// TIA Portal project "Inteligenta_szklarnia" (V15.1)

(* hardware
DEVICE "S7-1200 station_2"  S7-1200 Station
   slot 0: "Rack_0"  S7-1200 Rack  Rack  V1.0
   slot 1: "PLC_1"  CPU 1214C AC/DC/Rly  6ES7 214-1BE30-0XB0  V2.2
DEVICE "HMI_1"  KTP700 Basic PN
   slot 0: "HMI_1"  KTP700 Basic PN  6AV2 123-2GB03-0AX0  15.0.0.0
   slot 1: "HMI_RT_3"  KTP700 Basic PN  6AV2 123-2GB03-0AX0  15.0.0.0
   slot 5: "HMI_1.IE_CP_1"  PROFINET Interface  15.0.0.0
      slot 1: "PROFINET Interface_1"  PROFINET Interface
         slot 1: "Port_1"  Port
DEVICE "S7-1200 station_1"  S7-1200 Station
   slot 0: "Rack_0"  S7-1200 Rack  Rack  V1.0
   slot 1: "PLC_do_symulacji"  CPU 1214C AC/DC/Rly  6ES7 214-1BG40-0XB0  V4.2
DEVICE "HMI_do_symulacji"  KTP700 Basic PN
   slot 0: "HMI_do_symulacji"  KTP700 Basic PN  6AV2 123-2GB03-0AX0  15.1.0.0
   slot 1: "HMI_RT_2"  KTP700 Basic PN  6AV2 123-2GB03-0AX0  15.1.0.0
   slot 5: "HMI_do_symulacji.IE_CP_1"  PROFINET Interface  15.0.1.0
      slot 1: "PROFINET Interface_1"  PROFINET Interface
         slot 1: "Port_1"  Port
DEVICE "S71500/ET200MP station_1"  S7-1500 station
   slot 0: "Rail_0"  Rack  6ES7 590-1***0-0AA0
   slot 1: "PLC_Web_server"  CPU 1518-4 PN/DP  6ES7 518-4AP00-0AB0  V2.6
      slot 3: "CPU display_1"  6ES7591-1BA00-0AA0
*)

// ===== PLC "PLC_1"  CPU 1214C AC/DC/Rly =====

VAR_GLOBAL   // PLC tag table "Default tag table"
   "Tag_1" AT %M0.0 : Bool;
   "System_Byte" AT %MB1 : Byte;
   "FirstScan" AT %M1.0 : Bool;
   "DiagStatusUpdate" AT %M1.1 : Bool;
   "AlwaysTRUE" AT %M1.2 : Bool;
   "AlwaysFALSE" AT %M1.3 : Bool;
   "Tag_2" AT %M0.1 : Bool;
   "Clock_Byte" AT %MB30 : Byte;
   "Clock_10Hz" AT %M30.0 : Bool;
   "Clock_5Hz" AT %M30.1 : Bool;
   "Clock_2.5Hz" AT %M30.2 : Bool;
   "Clock_2Hz" AT %M30.3 : Bool;
   "Clock_1.25Hz" AT %M30.4 : Bool;
   "Clock_1Hz" AT %M30.5 : Bool;
   "Clock_0.625Hz" AT %M30.6 : Bool;
   "Clock_0.5Hz" AT %M30.7 : Bool;
   "marker_clock" AT %M0.2 : Bool;
   "marker_counter" AT %M0.3 : Bool;
   "wartosc_rolet_sym" AT %MW2 : Int;
   "swiatlo_bez_rolet" AT %MW4 : Int;
   "Alarm_active" AT %M8.0 : Bool;
   "Clock_Byte(1)" AT %MB0 : Byte;
   "Clock_10Hz(1)" AT %M0.0 : Bool;
   "Clock_5Hz(1)" AT %M0.1 : Bool;
   "Clock_2.5Hz(1)" AT %M0.2 : Bool;
   "Clock_2Hz(1)" AT %M0.3 : Bool;
   "Clock_1.25Hz(1)" AT %M0.4 : Bool;
   "Clock_1Hz(1)" AT %M0.5 : Bool;
   "Clock_0.625Hz(1)" AT %M0.6 : Bool;
   "Clock_0.5Hz(1)" AT %M0.7 : Bool;
END_VAR

VAR_GLOBAL   // PLC tag table "wyjscia"
   "Grzałka" AT %Q0.0 : Bool;
   "Wentylator" AT %Q0.1 : Bool;
   "Pompa_zraszacze" AT %Q0.2 : Bool;   // Pompa zraszaczy, które odpowiadają za wilgotność powietrza w szklarni
   "Rolety_zamykanie" AT %Q0.4 : Bool;
   "Alarm_ostrzegwaczy" AT %Q0.5 : Bool;
   "Siłownik_okien_otwieranie" AT %Q0.6 : Bool;
   "Siłownik_okien_zamykanie" AT %Q0.7 : Bool;
   "Rolety_otwieranie" AT %Q0.3 : Bool;
   "Pompa_podlewanie" AT %Q1.0 : Bool;   // Pompa podlewania kropelkowego, która odpowiada za wilgotność gleby
END_VAR

DATA_BLOCK "Wejscia_PLC"   // DB1
{ S7_Optimized_Access := 'TRUE' }
VERSION : 0.1
   VAR
      Czujnik_wilgotności_powietrza : Int;   // Czujnik wilgotności powietrza w szklarni
      Czujnik_wilgotności_gleby : Int;   // Czujnik wilgotności gleby w szklarni
      Temperatura_wewnetrzna : Real;   // Temperatura wewnątrz szklarni
      Czujnik_natezenia_swiatła : Int;   // Czujnik natężenia światła wewnątrz szklarni
      Czujnik_wiatru : Int;   // Czujnik prędkości wiatru poza szklarnią
      Wewnetrzny_czujnik_CO2 : Int;   // Czujnik stężenia dwutlenku węgla w szklarni
      Stopien_zasloniecia_rolet : Int;   // Stopień zasłonięcia rolet w szklarni (przyjęty przedział 0-100%)
      Temperatura_zewnetrzna : Real;   // Temperatura mierzona na zewnątrz, poza szklarnią. Typ Int, ponieważ nie jest wymagana taka dokładność jak w pomiarze temperatury wewnętrznej.
      Zewnetrzny_czujnik_CO2 : Int;   // Czujnik stężenia dwutlenku węgla poza szklarnią
      czujnik_wilgotnosci_zewnetrzny : Int := 50;   // Potrzebny w ramach symulacji realnych warunkow
   END_VAR
BEGIN
END_DATA_BLOCK

DATA_BLOCK "HMI"   // DB2
{ S7_Optimized_Access := 'TRUE' }
VERSION : 0.1
   VAR
      nazwa_receptury : String;
      System_okien_auto : Bool;   // Wł/wył system okien w trybie automatycznym
      Przycisk_zraszacze_manual : Bool;   // Przycisk pompy zraszaczy w trybie manualnym
      Przycisk_podlewanie_manual : Bool;   // Przycisk pompy podlewania w trybie manualnym
      Przycisk_grzanie_manual : Bool;   // Przycisk grzałki w trybie manualnym
      Przycisk_wentylacja_manual : Bool;   // Przycisk wentylacji w trybie manualnym
      Otwarcie_okien_manual : Bool;   // Ustawiony w trybie manualnym otwarcie okien
      Stopien_zasloniecia_rolet_manual : Int;   // Ustawiony w trybie manualnym stopień zasłonięcia rolet
      Temperatura_auto : Real := 22.0;   // Nastawiona temeratura w trybie automatycznym
      Naslonecznienie_auto : Int := 1000;   // Nastawiona wartość nasłonecznienia w trybie automatycznym
      Wilgotnosc_powietrza_auto : Int := 50;   // Nastawiona wartość wilgotności powietrza w trybie automatycznym
      Poziom_CO2_auto : Int := 800;   // Nastawiona wartość stężenia CO2 w trybie automatycznym
      Wilgotnosc_gleby_auto : Int := 60;   // Nastawiona wartość wilgotności gleby w trybie automatycznym
      Przycisk_zatwierdz_auto : Bool;   // Przycisk zatwierdzający wcześniej wybrane ustawienia trybu automatycznego
      Przycisk_zatwierdz_zapis_receptury : Bool;   // Przycisk zatwierdzający wcześniej wybrane ustawienia trybu zapisania receptury
      Przycisk_zatwierdz_wybor_receptury : Bool;   // Przycisk zatwierdzający wcześniej wybrane ustawienia trybu receptury
      Numer_ekranu_HMI : Int;   // Numer aktualnie otwartego ekranu w HMI
      Aktywacja_trybu_manualnego : Bool;
      Aktywacja_trybu_automatycznego : Bool;
      Aktywacja_trybu_Receptur : Bool;
      Aktywacja_trybu_zapis_Receptur : Bool;
      Reset_Trybow : Bool;
   END_VAR
BEGIN
END_DATA_BLOCK

DATA_BLOCK "Tryb_auto_parametry"   // DB7
{ S7_Optimized_Access := 'TRUE' }
VERSION : 0.1
   VAR
      Temperatura : Real;
      Naslonecznienie : Int;
      Wilgotnosc_powietrza : Int;
      Wilgotnosc_gleby : Int;
      System_okien : Bool;
      Stezenie_co2 : Int;
   END_VAR
BEGIN
END_DATA_BLOCK

DATA_BLOCK "Alarmy"   // DB9
{ S7_Optimized_Access := 'TRUE' }
VERSION : 0.1
   VAR
      Warning_niska_temp_1 : Bool;
      Warning_wysoka_temp_1 : Bool;
      Warning_nieprawidlowe_CO2_1 : Bool;
      Blad_zbyt_wysokie_CO2_1 : Bool;
   END_VAR
BEGIN
END_DATA_BLOCK

// folder: Archiwizacja_parametrow

DATA_BLOCK "Archiwizowane_parametry"   // DB4
{ S7_Optimized_Access := 'TRUE' }
VERSION : 0.1
   VAR
      Temperatura : Array[0..111] of Real;
      Wilgotnosc : Array[0..111] of Int;
      Naslonecznienie : Array[0..111] of Int;
      iterator : Int := 0;   // Iterator służący do zapisu danych w odpowiednich komórkach tablicy.
   END_VAR
BEGIN
   Naslonecznienie[0] := 0;
   Naslonecznienie[1] := 0;
END_DATA_BLOCK

// folder: System blocks/Program resources

DATA_BLOCK "IEC_Counter_0_DB_1"   // DB3
{ S7_Optimized_Access := 'TRUE' }
AUTHOR : Simatic
FAMILY : IEC
NAME : CNTR
VERSION : 1.0
// stored: InstanceOfName IEC_COUNTER
"IEC_COUNTER"
BEGIN
END_DATA_BLOCK

DATA_BLOCK "IEC_Timer_0_DB"   // DB5
{ S7_Optimized_Access := 'TRUE' }
AUTHOR : Simatic
FAMILY : IEC
NAME : IEC_TMR
VERSION : 1.0
// stored: InstanceOfName IEC_TIMER
"IEC_TIMER"
BEGIN
END_DATA_BLOCK

DATA_BLOCK "IEC_Timer_0_DB_1"   // DB6
{ S7_Optimized_Access := 'TRUE' }
AUTHOR : Simatic
FAMILY : IEC
NAME : IEC_TMR
VERSION : 1.0
// stored: InstanceOfName IEC_TIMER
"IEC_TIMER"
BEGIN
END_DATA_BLOCK

DATA_BLOCK "IEC_Timer_0_DB_2"   // DB8
{ S7_Optimized_Access := 'TRUE' }
AUTHOR : Simatic
FAMILY : IEC
NAME : IEC_TMR
VERSION : 1.0
// stored: InstanceOfName IEC_TIMER
"IEC_TIMER"
BEGIN
END_DATA_BLOCK

DATA_BLOCK "IEC_Timer_0_DB_5"   // DB10
{ S7_Optimized_Access := 'TRUE' }
AUTHOR : Simatic
FAMILY : IEC
NAME : IEC_TMR
VERSION : 1.0
// stored: InstanceOfName IEC_TIMER
"IEC_TIMER"
BEGIN
END_DATA_BLOCK

DATA_BLOCK "IEC_Timer_0_DB_3"   // DB11
{ S7_Optimized_Access := 'TRUE' }
AUTHOR : Simatic
FAMILY : IEC
NAME : IEC_TMR
VERSION : 1.0
// stored: InstanceOfName IEC_TIMER
"IEC_TIMER"
BEGIN
END_DATA_BLOCK

DATA_BLOCK "IEC_Counter_0_DB"   // DB12
{ S7_Optimized_Access := 'TRUE' }
AUTHOR : Simatic
FAMILY : IEC
NAME : CNTR
VERSION : 1.0
// stored: InstanceOfName IEC_COUNTER
"IEC_COUNTER"
BEGIN
END_DATA_BLOCK

DATA_BLOCK "IEC_Counter_0_DB_2"   // DB13
{ S7_Optimized_Access := 'TRUE' }
AUTHOR : Simatic
FAMILY : IEC
NAME : CNTR
VERSION : 1.0
// stored: InstanceOfName IEC_COUNTER
"IEC_COUNTER"
BEGIN
END_DATA_BLOCK

// folder: (top level)

FUNCTION "Rolety" : Void   // FC1, LAD
{ S7_Optimized_Access := 'TRUE' }
VERSION : 0.1
   VAR_INPUT
      Czy_automatyczny : Bool;
      Czy_manualny : Bool;
   END_VAR
BEGIN

REGION Network 1: Warunki otwierania rolet w trybie automatycznym i manualnym
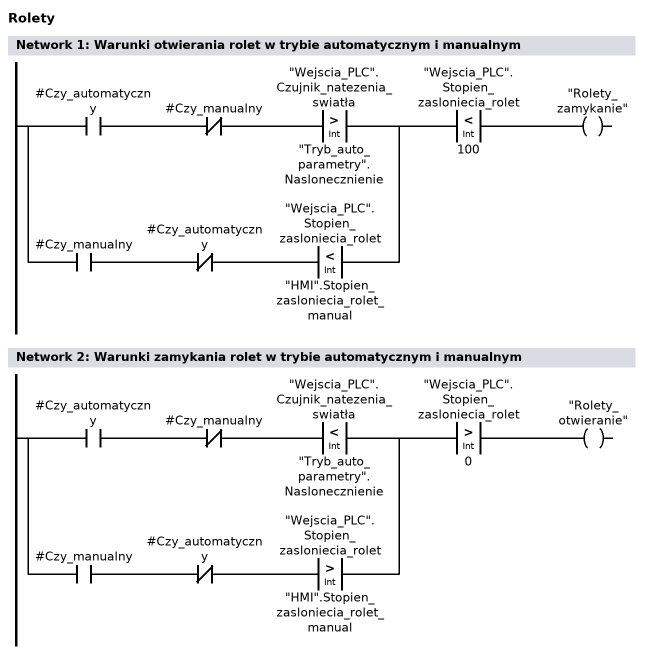
   RUNG wire#powerrail
      Contact( #Czy_automatyczny )
      I_Contact( #Czy_manualny )
      { S7_Templates := "SrcType := Int" } GT_Contact(in1 := "Wejscia_PLC".Czujnik_natezenia_swiatła, in2 := "Tryb_auto_parametry".Naslonecznienie)
      wire#w1
      { S7_Templates := "SrcType := Int" } LT_Contact(in1 := "Wejscia_PLC".Stopien_zasloniecia_rolet, in2 := 100)
      Coil( "Rolety_zamykanie" )
   END_RUNG
   RUNG wire#powerrail
      Contact( #Czy_manualny )
      I_Contact( #Czy_automatyczny )
      { S7_Templates := "SrcType := Int" } LT_Contact(in1 := "Wejscia_PLC".Stopien_zasloniecia_rolet, in2 := "HMI".Stopien_zasloniecia_rolet_manual)
   END_RUNG wire#w1
   // the same network as SCL:
   "Rolety_zamykanie" := ((#Czy_automatyczny AND NOT #Czy_manualny AND ("Wejscia_PLC".Czujnik_natezenia_swiatła > "Tryb_auto_parametry".Naslonecznienie)) OR (#Czy_manualny AND NOT #Czy_automatyczny AND ("Wejscia_PLC".Stopien_zasloniecia_rolet < "HMI".Stopien_zasloniecia_rolet_manual))) AND ("Wejscia_PLC".Stopien_zasloniecia_rolet < 100);
END_REGION

REGION Network 2: Warunki zamykania rolet w trybie automatycznym i manualnym
   RUNG wire#powerrail
      Contact( #Czy_automatyczny )
      I_Contact( #Czy_manualny )
      { S7_Templates := "SrcType := Int" } LT_Contact(in1 := "Wejscia_PLC".Czujnik_natezenia_swiatła, in2 := "Tryb_auto_parametry".Naslonecznienie)
      wire#w1
      { S7_Templates := "SrcType := Int" } GT_Contact(in1 := "Wejscia_PLC".Stopien_zasloniecia_rolet, in2 := 0)
      Coil( "Rolety_otwieranie" )
   END_RUNG
   RUNG wire#powerrail
      Contact( #Czy_manualny )
      I_Contact( #Czy_automatyczny )
      { S7_Templates := "SrcType := Int" } GT_Contact(in1 := "Wejscia_PLC".Stopien_zasloniecia_rolet, in2 := "HMI".Stopien_zasloniecia_rolet_manual)
   END_RUNG wire#w1
   // the same network as SCL:
   "Rolety_otwieranie" := ((#Czy_automatyczny AND NOT #Czy_manualny AND ("Wejscia_PLC".Czujnik_natezenia_swiatła < "Tryb_auto_parametry".Naslonecznienie)) OR (#Czy_manualny AND NOT #Czy_automatyczny AND ("Wejscia_PLC".Stopien_zasloniecia_rolet > "HMI".Stopien_zasloniecia_rolet_manual))) AND ("Wejscia_PLC".Stopien_zasloniecia_rolet > 0);
END_REGION
END_FUNCTION

FUNCTION "Sterowanie_grzalka_wentylator" : Void   // FC3, LAD
{ S7_Optimized_Access := 'TRUE' }
VERSION : 0.1
   VAR_INPUT
      czy_manualny : Bool;
      czy_automatyczny : Bool;
   END_VAR
   VAR_TEMP
      Histereza_minus : Real;   // Wartość zadanej temperatury zmieniona o dolną wartość hiterezy
      Histereza_plus : Real;   // Wartość zadanej temperatury zmieniona o górną wartość hiterezy
   END_VAR
   VAR CONSTANT
      Wartosc_histerezy : Real := 1.0;
   END_VAR
   VAR_TEMP   // added for the SCL form of the ladder/FBD networks
      _w1 : Bool;
   END_VAR
BEGIN

REGION Network 1: Sterowanie wentylatorem w trybie automatycznym i manualnym
   // Gdy uruchomiony jest tryb automatyczny, wartość temperatury w szklarni powinna się mieścić w zakresie temperatury nastawionej +- wartość histerezy. Gdy jest ona za wysoka uruchamiany jest wentylator. W trybie manualnym włączany jest on od razu po naciśnięciu przycisku do niego przypisanego.
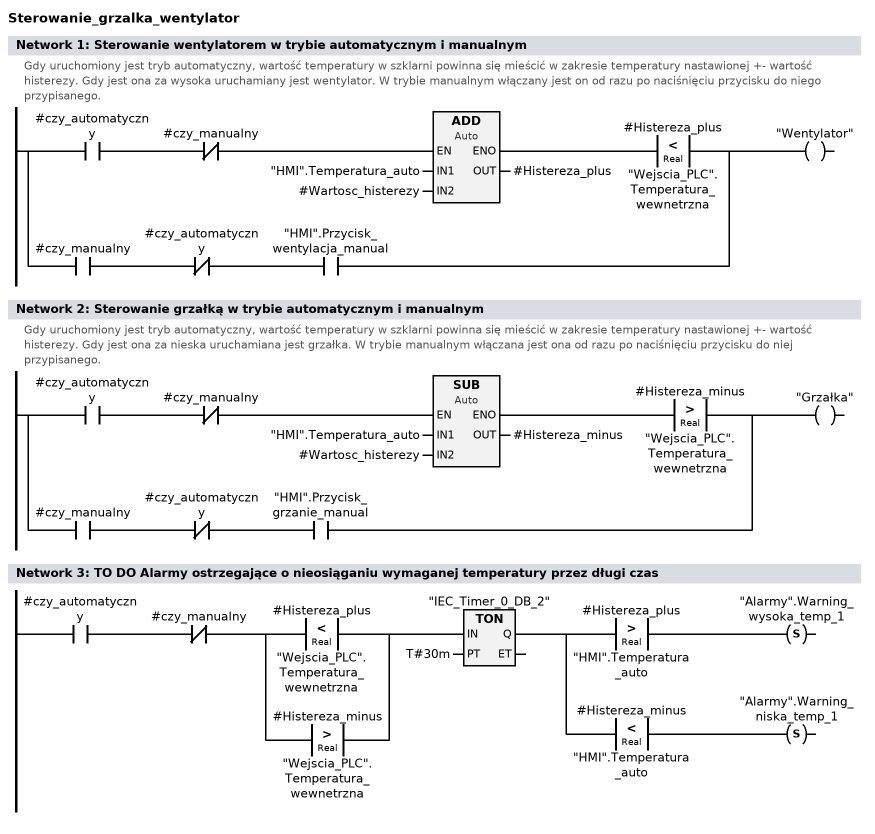
   RUNG wire#powerrail
      Contact( #czy_automatyczny )
      I_Contact( #czy_manualny )
      { S7_GenerateENO := "TRUE" } Add(in1 := "HMI".Temperatura_auto, in2 := #Wartosc_histerezy, out => #Histereza_plus)
      { S7_Templates := "SrcType := Real" } LT_Contact(in1 := #Histereza_plus, in2 := "Wejscia_PLC".Temperatura_wewnetrzna)
      wire#w1
      Coil( "Wentylator" )
   END_RUNG
   RUNG wire#powerrail
      Contact( #czy_manualny )
      I_Contact( #czy_automatyczny )
      Contact( "HMI".Przycisk_wentylacja_manual )
   END_RUNG wire#w1
   // the same network as SCL:
   // ENO of a box is taken as its EN; it also drops when the box reports an error
   #_w1 := #czy_automatyczny AND NOT #czy_manualny;
   IF #_w1 THEN #Histereza_plus := "HMI".Temperatura_auto + #Wartosc_histerezy; END_IF;
   "Wentylator" := (#_w1 AND (#Histereza_plus < "Wejscia_PLC".Temperatura_wewnetrzna)) OR (#czy_manualny AND NOT #czy_automatyczny AND "HMI".Przycisk_wentylacja_manual);
END_REGION

REGION Network 2: Sterowanie grzałką w trybie automatycznym i manualnym
   // Gdy uruchomiony jest tryb automatyczny, wartość temperatury w szklarni powinna się mieścić w zakresie temperatury nastawionej +- wartość histerezy. Gdy jest ona za nieska uruchamiana jest grzałka. W trybie manualnym włączana jest ona od razu po naciśnięciu przycisku do niej przypisanego.
   RUNG wire#powerrail
      Contact( #czy_automatyczny )
      I_Contact( #czy_manualny )
      { S7_GenerateENO := "TRUE" } Sub(in1 := "HMI".Temperatura_auto, in2 := #Wartosc_histerezy, out => #Histereza_minus)
      { S7_Templates := "SrcType := Real" } GT_Contact(in1 := #Histereza_minus, in2 := "Wejscia_PLC".Temperatura_wewnetrzna)
      wire#w1
      Coil( "Grzałka" )
   END_RUNG
   RUNG wire#powerrail
      Contact( #czy_manualny )
      I_Contact( #czy_automatyczny )
      Contact( "HMI".Przycisk_grzanie_manual )
   END_RUNG wire#w1
   // the same network as SCL:
   // ENO of a box is taken as its EN; it also drops when the box reports an error
   #_w1 := #czy_automatyczny AND NOT #czy_manualny;
   IF #_w1 THEN #Histereza_minus := "HMI".Temperatura_auto - #Wartosc_histerezy; END_IF;
   "Grzałka" := (#_w1 AND (#Histereza_minus > "Wejscia_PLC".Temperatura_wewnetrzna)) OR (#czy_manualny AND NOT #czy_automatyczny AND "HMI".Przycisk_grzanie_manual);
END_REGION

REGION Network 3: TO DO Alarmy ostrzegające o nieosiąganiu wymaganej temperatury przez długi czas
   "IEC_Timer_0_DB_2".TON(IN := #czy_automatyczny AND NOT #czy_manualny AND ((#Histereza_plus < "Wejscia_PLC".Temperatura_wewnetrzna) OR (#Histereza_minus > "Wejscia_PLC".Temperatura_wewnetrzna)),
                          PT := T#30m);
   IF "IEC_Timer_0_DB_2".Q AND (#Histereza_plus > "HMI".Temperatura_auto) THEN
       "Alarmy".Warning_wysoka_temp_1 := TRUE;
   END_IF;
   IF "IEC_Timer_0_DB_2".Q AND (#Histereza_minus < "HMI".Temperatura_auto) THEN
       "Alarmy".Warning_niska_temp_1 := TRUE;
   END_IF;
END_REGION
END_FUNCTION

FUNCTION "Zapis_parametrow_trybu_auto" : Void   // FC4, LAD
{ S7_Optimized_Access := 'TRUE' }
VERSION : 0.1
BEGIN

REGION Network 1: Zapis wybranych na HMI parametrów, aby zostały one stałe do kolejnego zatwierdzenia ich zmiany.
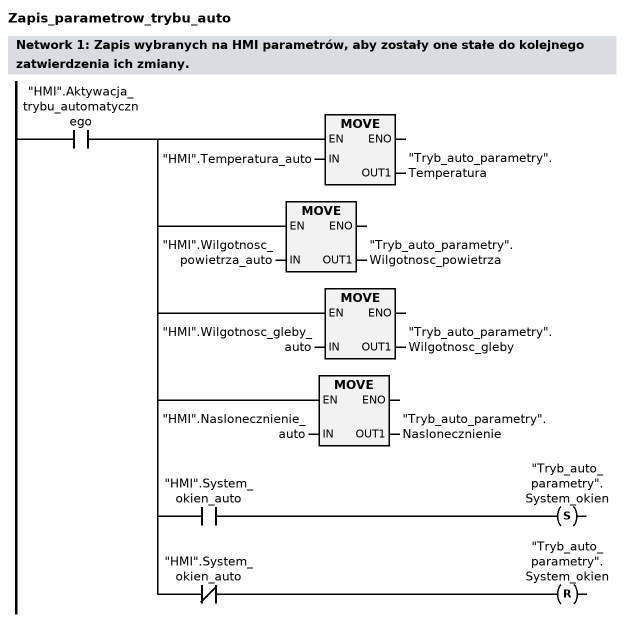
   RUNG wire#powerrail
      Contact( "HMI".Aktywacja_trybu_automatycznego )
      wire#w1
      { S7_GenerateENO := "TRUE" } Move(in := "HMI".Temperatura_auto, out1 => "Tryb_auto_parametry".Temperatura)
   END_RUNG
   RUNG wire#w1
      { S7_GenerateENO := "TRUE" } Move(in := "HMI".Wilgotnosc_powietrza_auto, out1 => "Tryb_auto_parametry".Wilgotnosc_powietrza)
   END_RUNG
   RUNG wire#w1
      { S7_GenerateENO := "TRUE" } Move(in := "HMI".Wilgotnosc_gleby_auto, out1 => "Tryb_auto_parametry".Wilgotnosc_gleby)
   END_RUNG
   RUNG wire#w1
      { S7_GenerateENO := "TRUE" } Move(in := "HMI".Naslonecznienie_auto, out1 => "Tryb_auto_parametry".Naslonecznienie)
   END_RUNG
   RUNG wire#w1
      Contact( "HMI".System_okien_auto )
      S_Coil( "Tryb_auto_parametry".System_okien )
   END_RUNG
   RUNG wire#w1
      I_Contact( "HMI".System_okien_auto )
      R_Coil( "Tryb_auto_parametry".System_okien )
   END_RUNG
   // the same network as SCL:
   IF "HMI".Aktywacja_trybu_automatycznego THEN
       "Tryb_auto_parametry".Temperatura := "HMI".Temperatura_auto;
       "Tryb_auto_parametry".Wilgotnosc_powietrza := "HMI".Wilgotnosc_powietrza_auto;
       "Tryb_auto_parametry".Wilgotnosc_gleby := "HMI".Wilgotnosc_gleby_auto;
       "Tryb_auto_parametry".Naslonecznienie := "HMI".Naslonecznienie_auto;
   END_IF;
   IF "HMI".Aktywacja_trybu_automatycznego AND "HMI".System_okien_auto THEN
       "Tryb_auto_parametry".System_okien := TRUE;
   END_IF;
   IF "HMI".Aktywacja_trybu_automatycznego AND NOT "HMI".System_okien_auto THEN
       "Tryb_auto_parametry".System_okien := FALSE;
   END_IF;
END_REGION
END_FUNCTION

FUNCTION "Jaki_Tryb" : Void   // FC5, LAD
{ S7_Optimized_Access := 'TRUE' }
VERSION : 0.1
BEGIN

REGION Network 1: Reset trybu auto jesli wykryje jakikolwiek inny tryb
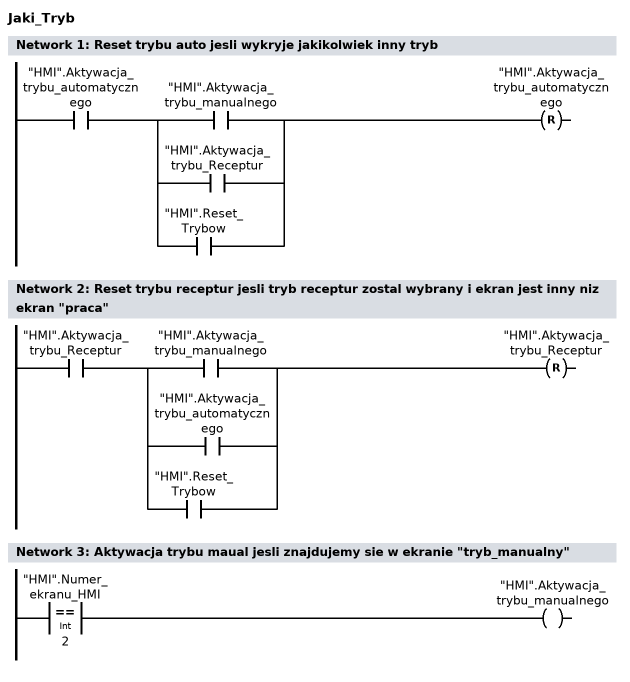
   RUNG wire#powerrail
      Contact( "HMI".Aktywacja_trybu_automatycznego )
      wire#w1
      Contact( "HMI".Aktywacja_trybu_manualnego )
      wire#w2
      R_Coil( "HMI".Aktywacja_trybu_automatycznego )
   END_RUNG
   RUNG wire#w1
      Contact( "HMI".Aktywacja_trybu_Receptur )
   END_RUNG wire#w2
   RUNG wire#w1
      Contact( "HMI".Reset_Trybow )
   END_RUNG wire#w2
   // the same network as SCL:
   IF "HMI".Aktywacja_trybu_automatycznego AND ("HMI".Aktywacja_trybu_manualnego OR "HMI".Aktywacja_trybu_Receptur OR "HMI".Reset_Trybow) THEN
       "HMI".Aktywacja_trybu_automatycznego := FALSE;
   END_IF;
END_REGION

REGION Network 2: Reset trybu receptur jesli tryb receptur zostal wybrany i ekran jest inny niz ekran "praca"
   RUNG wire#powerrail
      Contact( "HMI".Aktywacja_trybu_Receptur )
      wire#w1
      Contact( "HMI".Aktywacja_trybu_manualnego )
      wire#w2
      R_Coil( "HMI".Aktywacja_trybu_Receptur )
   END_RUNG
   RUNG wire#w1
      Contact( "HMI".Aktywacja_trybu_automatycznego )
   END_RUNG wire#w2
   RUNG wire#w1
      Contact( "HMI".Reset_Trybow )
   END_RUNG wire#w2
   // the same network as SCL:
   IF "HMI".Aktywacja_trybu_Receptur AND ("HMI".Aktywacja_trybu_manualnego OR "HMI".Aktywacja_trybu_automatycznego OR "HMI".Reset_Trybow) THEN
       "HMI".Aktywacja_trybu_Receptur := FALSE;
   END_IF;
END_REGION

REGION Network 3: Aktywacja trybu maual jesli znajdujemy sie w ekranie "tryb_manualny"
   RUNG wire#powerrail
      { S7_Templates := "SrcType := Int" } EQ_Contact(in1 := "HMI".Numer_ekranu_HMI, in2 := 2)
      Coil( "HMI".Aktywacja_trybu_manualnego )
   END_RUNG
   // the same network as SCL:
   "HMI".Aktywacja_trybu_manualnego := "HMI".Numer_ekranu_HMI = 2;
END_REGION
END_FUNCTION

FUNCTION "Ograniczanie_wartosci_parametrow" : Void   // FC6, LAD
TITLE = Każdy z poniższych network-ów odpowiada za to, aby po ustawieniu na HMI wartości przekraczajacej dopuszczalną, ta pozostała w wymaganym zakresie.
{ S7_Optimized_Access := 'TRUE' }
VERSION : 0.1
BEGIN

REGION Network 1: Ograniczenie dla wartosci ustawionej temperatury w trybie automatycznym
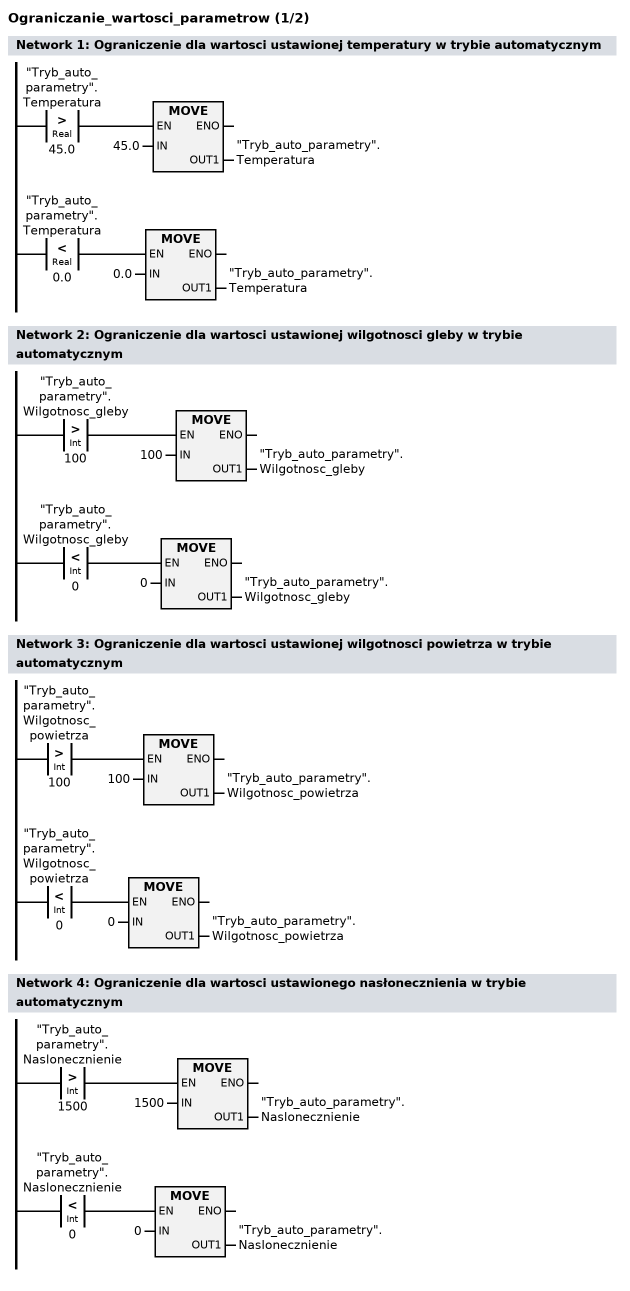
   RUNG wire#powerrail
      { S7_Templates := "SrcType := Real" } GT_Contact(in1 := "Tryb_auto_parametry".Temperatura, in2 := 45.0)
      { S7_GenerateENO := "TRUE" } Move(in := 45.0, out1 => "Tryb_auto_parametry".Temperatura)
   END_RUNG
   RUNG wire#powerrail
      { S7_Templates := "SrcType := Real" } LT_Contact(in1 := "Tryb_auto_parametry".Temperatura, in2 := 0.0)
      { S7_GenerateENO := "TRUE" } Move(in := 0.0, out1 => "Tryb_auto_parametry".Temperatura)
   END_RUNG
   // the same network as SCL:
   IF "Tryb_auto_parametry".Temperatura > 45.0 THEN "Tryb_auto_parametry".Temperatura := 45.0; END_IF;
   IF "Tryb_auto_parametry".Temperatura < 0.0 THEN "Tryb_auto_parametry".Temperatura := 0.0; END_IF;
END_REGION

REGION Network 2: Ograniczenie dla wartosci ustawionej wilgotnosci gleby w trybie automatycznym
   RUNG wire#powerrail
      { S7_Templates := "SrcType := Int" } GT_Contact(in1 := "Tryb_auto_parametry".Wilgotnosc_gleby, in2 := 100)
      { S7_GenerateENO := "TRUE" } Move(in := 100, out1 => "Tryb_auto_parametry".Wilgotnosc_gleby)
   END_RUNG
   RUNG wire#powerrail
      { S7_Templates := "SrcType := Int" } LT_Contact(in1 := "Tryb_auto_parametry".Wilgotnosc_gleby, in2 := 0)
      { S7_GenerateENO := "TRUE" } Move(in := 0, out1 => "Tryb_auto_parametry".Wilgotnosc_gleby)
   END_RUNG
   // the same network as SCL:
   IF "Tryb_auto_parametry".Wilgotnosc_gleby > 100 THEN
       "Tryb_auto_parametry".Wilgotnosc_gleby := 100;
   END_IF;
   IF "Tryb_auto_parametry".Wilgotnosc_gleby < 0 THEN "Tryb_auto_parametry".Wilgotnosc_gleby := 0; END_IF;
END_REGION

REGION Network 3: Ograniczenie dla wartosci ustawionej wilgotnosci powietrza w trybie automatycznym
   RUNG wire#powerrail
      { S7_Templates := "SrcType := Int" } GT_Contact(in1 := "Tryb_auto_parametry".Wilgotnosc_powietrza, in2 := 100)
      { S7_GenerateENO := "TRUE" } Move(in := 100, out1 => "Tryb_auto_parametry".Wilgotnosc_powietrza)
   END_RUNG
   RUNG wire#powerrail
      { S7_Templates := "SrcType := Int" } LT_Contact(in1 := "Tryb_auto_parametry".Wilgotnosc_powietrza, in2 := 0)
      { S7_GenerateENO := "TRUE" } Move(in := 0, out1 => "Tryb_auto_parametry".Wilgotnosc_powietrza)
   END_RUNG
   // the same network as SCL:
   IF "Tryb_auto_parametry".Wilgotnosc_powietrza > 100 THEN
       "Tryb_auto_parametry".Wilgotnosc_powietrza := 100;
   END_IF;
   IF "Tryb_auto_parametry".Wilgotnosc_powietrza < 0 THEN
       "Tryb_auto_parametry".Wilgotnosc_powietrza := 0;
   END_IF;
END_REGION

REGION Network 4: Ograniczenie dla wartosci ustawionego nasłonecznienia w trybie automatycznym
   RUNG wire#powerrail
      { S7_Templates := "SrcType := Int" } GT_Contact(in1 := "Tryb_auto_parametry".Naslonecznienie, in2 := 1500)
      { S7_GenerateENO := "TRUE" } Move(in := 1500, out1 => "Tryb_auto_parametry".Naslonecznienie)
   END_RUNG
   RUNG wire#powerrail
      { S7_Templates := "SrcType := Int" } LT_Contact(in1 := "Tryb_auto_parametry".Naslonecznienie, in2 := 0)
      { S7_GenerateENO := "TRUE" } Move(in := 0, out1 => "Tryb_auto_parametry".Naslonecznienie)
   END_RUNG
   // the same network as SCL:
   IF "Tryb_auto_parametry".Naslonecznienie > 1500 THEN
       "Tryb_auto_parametry".Naslonecznienie := 1500;
   END_IF;
   IF "Tryb_auto_parametry".Naslonecznienie < 0 THEN "Tryb_auto_parametry".Naslonecznienie := 0; END_IF;
END_REGION

REGION Network 5: Ograniczenie dla wartosci ustawionego stężenia CO2 w trybie automatycznym
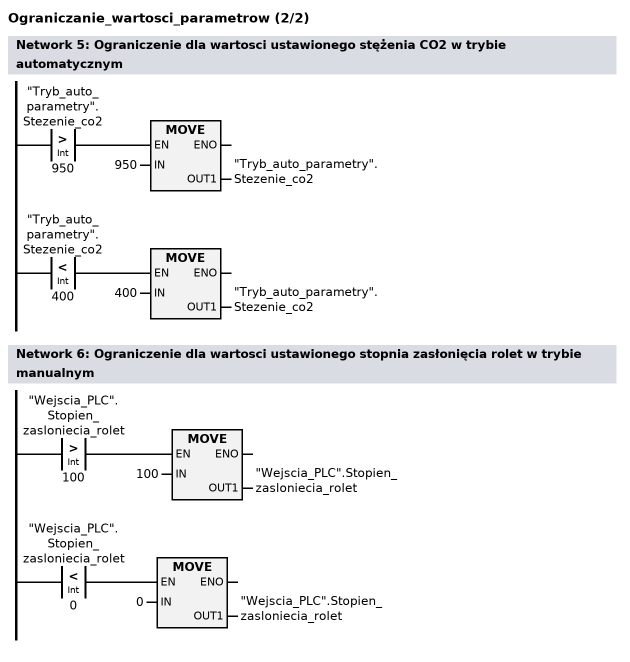
   RUNG wire#powerrail
      { S7_Templates := "SrcType := Int" } GT_Contact(in1 := "Tryb_auto_parametry".Stezenie_co2, in2 := 950)
      { S7_GenerateENO := "TRUE" } Move(in := 950, out1 => "Tryb_auto_parametry".Stezenie_co2)
   END_RUNG
   RUNG wire#powerrail
      { S7_Templates := "SrcType := Int" } LT_Contact(in1 := "Tryb_auto_parametry".Stezenie_co2, in2 := 400)
      { S7_GenerateENO := "TRUE" } Move(in := 400, out1 => "Tryb_auto_parametry".Stezenie_co2)
   END_RUNG
   // the same network as SCL:
   IF "Tryb_auto_parametry".Stezenie_co2 > 950 THEN "Tryb_auto_parametry".Stezenie_co2 := 950; END_IF;
   IF "Tryb_auto_parametry".Stezenie_co2 < 400 THEN "Tryb_auto_parametry".Stezenie_co2 := 400; END_IF;
END_REGION

REGION Network 6: Ograniczenie dla wartosci ustawionego stopnia zasłonięcia rolet w trybie manualnym
   RUNG wire#powerrail
      { S7_Templates := "SrcType := Int" } GT_Contact(in1 := "Wejscia_PLC".Stopien_zasloniecia_rolet, in2 := 100)
      { S7_GenerateENO := "TRUE" } Move(in := 100, out1 => "Wejscia_PLC".Stopien_zasloniecia_rolet)
   END_RUNG
   RUNG wire#powerrail
      { S7_Templates := "SrcType := Int" } LT_Contact(in1 := "Wejscia_PLC".Stopien_zasloniecia_rolet, in2 := 0)
      { S7_GenerateENO := "TRUE" } Move(in := 0, out1 => "Wejscia_PLC".Stopien_zasloniecia_rolet)
   END_RUNG
   // the same network as SCL:
   IF "Wejscia_PLC".Stopien_zasloniecia_rolet > 100 THEN
       "Wejscia_PLC".Stopien_zasloniecia_rolet := 100;
   END_IF;
   IF "Wejscia_PLC".Stopien_zasloniecia_rolet < 0 THEN "Wejscia_PLC".Stopien_zasloniecia_rolet := 0; END_IF;
END_REGION
END_FUNCTION

FUNCTION "Sterowanie_podlewaniem_zraszaniem" : Void   // FC7, LAD
{ S7_Optimized_Access := 'TRUE' }
VERSION : 0.1
   VAR_INPUT
      Czy_automatyczny : Bool;
      Czy_manualny : Bool;
   END_VAR
BEGIN

REGION Network 1: Sterowanie pompą zraszaczy, które odpowiadają za wilgotność powietrza w szklarni
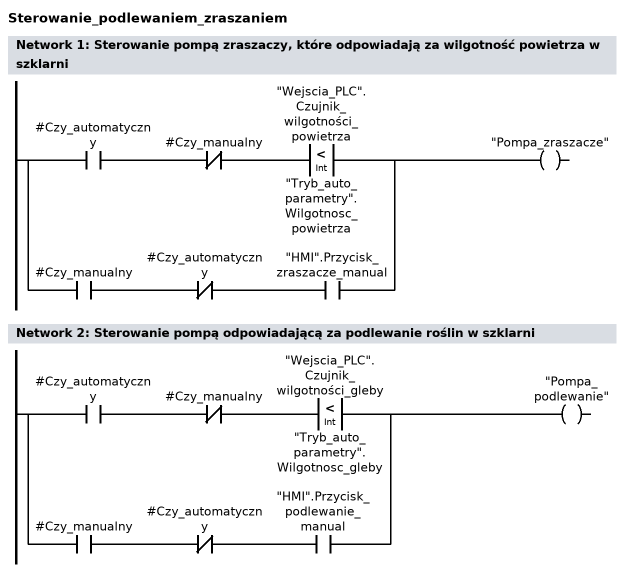
   RUNG wire#powerrail
      Contact( #Czy_automatyczny )
      I_Contact( #Czy_manualny )
      { S7_Templates := "SrcType := Int" } LT_Contact(in1 := "Wejscia_PLC".Czujnik_wilgotności_powietrza, in2 := "Tryb_auto_parametry".Wilgotnosc_powietrza)
      wire#w1
      Coil( "Pompa_zraszacze" )
   END_RUNG
   RUNG wire#powerrail
      Contact( #Czy_manualny )
      I_Contact( #Czy_automatyczny )
      Contact( "HMI".Przycisk_zraszacze_manual )
   END_RUNG wire#w1
   // the same network as SCL:
   "Pompa_zraszacze" := (#Czy_automatyczny AND NOT #Czy_manualny AND ("Wejscia_PLC".Czujnik_wilgotności_powietrza < "Tryb_auto_parametry".Wilgotnosc_powietrza)) OR (#Czy_manualny AND NOT #Czy_automatyczny AND "HMI".Przycisk_zraszacze_manual);
END_REGION

REGION Network 2: Sterowanie pompą odpowiadającą za podlewanie roślin w szklarni
   RUNG wire#powerrail
      Contact( #Czy_automatyczny )
      I_Contact( #Czy_manualny )
      { S7_Templates := "SrcType := Int" } LT_Contact(in1 := "Wejscia_PLC".Czujnik_wilgotności_gleby, in2 := "Tryb_auto_parametry".Wilgotnosc_gleby)
      wire#w1
      Coil( "Pompa_podlewanie" )
   END_RUNG
   RUNG wire#powerrail
      Contact( #Czy_manualny )
      I_Contact( #Czy_automatyczny )
      Contact( "HMI".Przycisk_podlewanie_manual )
   END_RUNG wire#w1
   // the same network as SCL:
   "Pompa_podlewanie" := (#Czy_automatyczny AND NOT #Czy_manualny AND ("Wejscia_PLC".Czujnik_wilgotności_gleby < "Tryb_auto_parametry".Wilgotnosc_gleby)) OR (#Czy_manualny AND NOT #Czy_automatyczny AND "HMI".Przycisk_podlewanie_manual);
END_REGION
END_FUNCTION

FUNCTION "Sterowanie_oknami" : Void   // FC8, LAD
{ S7_Optimized_Access := 'TRUE' }
VERSION : 0.1
   VAR_INPUT
      czy_manualny : Bool;
      czy_automatyczny : Bool;
   END_VAR
   VAR_TEMP
      Histereza_plus : Int;
      Histereza_minus : Int;
      Zakres_temp_gora : Real;   // Górny zakres temperatury zewnętrznej dla której w trybie automatycznym będą otwierane okna
      Zakres_temp_dol : Real;   // Dolny zakres temperatury zewnętrznej dla której w trybie automatycznym będą otwierane okna
   END_VAR
   VAR CONSTANT
      Histereza : Int := 25;   // Histereza, która określa kiedy stan CO2 w szklarni jest uznawany za prawidłowy
   END_VAR
BEGIN

REGION Network 1: Operacje matematyczne używane w networku 2. i 3.
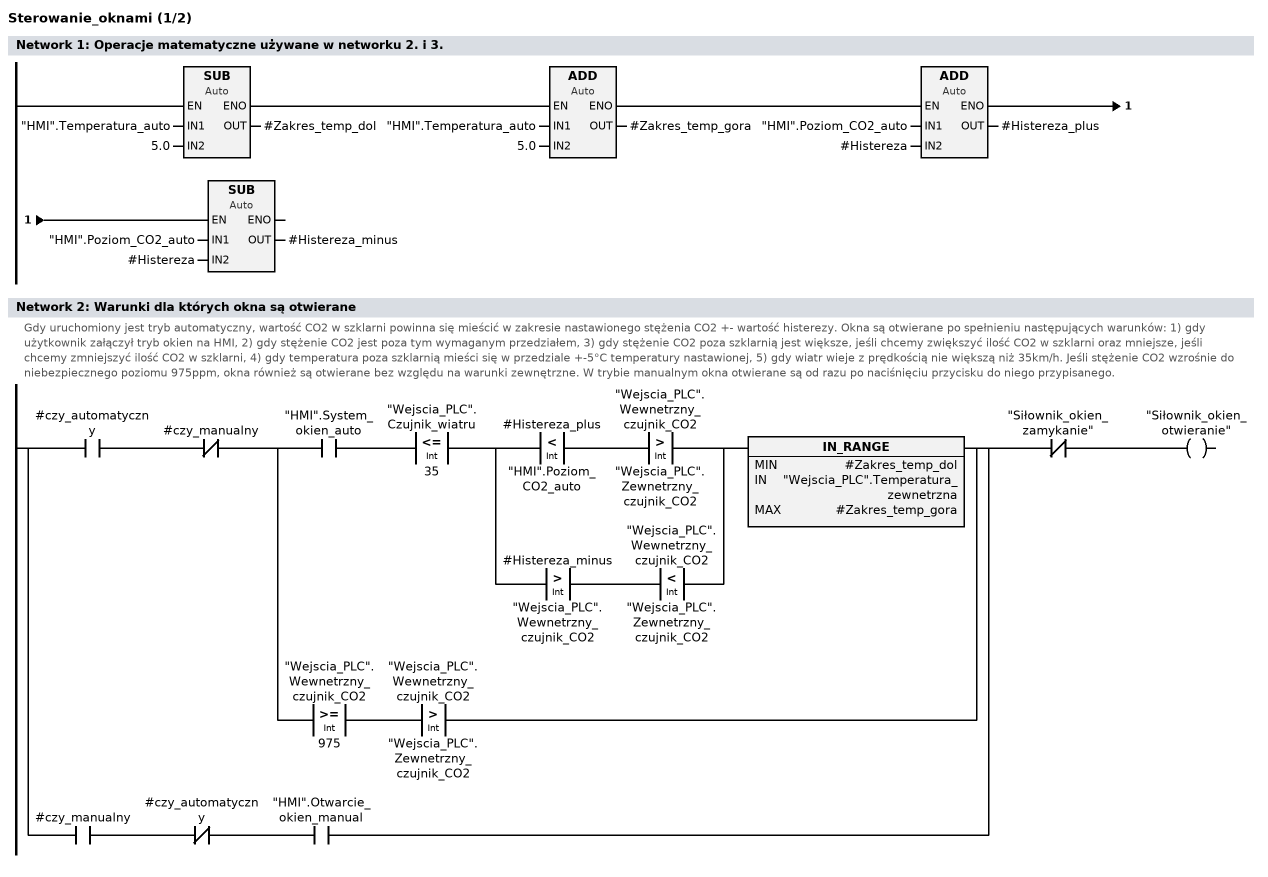
   RUNG wire#powerrail
      { S7_GenerateENO := "TRUE" } Sub(in1 := "HMI".Temperatura_auto, in2 := 5.0, out => #Zakres_temp_dol)
      { S7_GenerateENO := "TRUE" } Add(in1 := "HMI".Temperatura_auto, in2 := 5.0, out => #Zakres_temp_gora)
      { S7_GenerateENO := "TRUE" } Add(in1 := "HMI".Poziom_CO2_auto, in2 := #Histereza, out => #Histereza_plus)
      { S7_GenerateENO := "TRUE" } Sub(in1 := "HMI".Poziom_CO2_auto, in2 := #Histereza, out => #Histereza_minus)
   END_RUNG
   // the same network as SCL:
   // ENO of a box is taken as its EN; it also drops when the box reports an error
   #Zakres_temp_dol := "HMI".Temperatura_auto - 5.0;
   #Zakres_temp_gora := "HMI".Temperatura_auto + 5.0;
   #Histereza_plus := "HMI".Poziom_CO2_auto + #Histereza;
   #Histereza_minus := "HMI".Poziom_CO2_auto - #Histereza;
END_REGION

REGION Network 2: Warunki dla których okna są otwierane
   // Gdy uruchomiony jest tryb automatyczny, wartość CO2 w szklarni powinna się mieścić w zakresie nastawionego stężenia CO2 +- wartość histerezy. Okna są otwierane po spełnieniu następujących warunków: 1) gdy użytkownik załączył tryb okien na HMI, 2) gdy stężenie CO2 jest poza tym wymaganym przedziałem, 3) gdy stężenie CO2 poza szklarnią jest większe, jeśli chcemy zwiększyć ilość CO2 w szklarni oraz mniejsze, jeśli chcemy zmniejszyć ilość CO2 w szklarni, 4) gdy temperatura poza szklarnią mieści się w przedziale +-5°C temperatury nastawionej, 5) gdy wiatr wieje z prędkością nie większą niż 35km/h. Jeśli stężenie CO2 wzrośnie do niebezpiecznego poziomu 975ppm, okna również są otwierane bez względu na warunki zewnętrzne. W trybie manualnym okna otwierane są od razu po naciśnięciu przycisku do niego przypisanego.
   RUNG wire#powerrail
      Contact( #czy_automatyczny )
      I_Contact( #czy_manualny )
      wire#w1
      Contact( "HMI".System_okien_auto )
      { S7_Templates := "SrcType := Int" } LE_Contact(in1 := "Wejscia_PLC".Czujnik_wiatru, in2 := 35)
      wire#w2
      { S7_Templates := "SrcType := Int" } LT_Contact(in1 := #Histereza_plus, in2 := "HMI".Poziom_CO2_auto)
      { S7_Templates := "SrcType := Int" } GT_Contact(in1 := "Wejscia_PLC".Wewnetrzny_czujnik_CO2, in2 := "Wejscia_PLC".Zewnetrzny_czujnik_CO2)
      wire#w3
      { S7_Templates := "SrcType := Real" } InRange(min := #Zakres_temp_dol, in := "Wejscia_PLC".Temperatura_zewnetrzna, max := #Zakres_temp_gora)
      wire#w4
      I_Contact( "Siłownik_okien_zamykanie" )
      Coil( "Siłownik_okien_otwieranie" )
   END_RUNG
   RUNG wire#w2
      { S7_Templates := "SrcType := Int" } GT_Contact(in1 := #Histereza_minus, in2 := "Wejscia_PLC".Wewnetrzny_czujnik_CO2)
      { S7_Templates := "SrcType := Int" } LT_Contact(in1 := "Wejscia_PLC".Wewnetrzny_czujnik_CO2, in2 := "Wejscia_PLC".Zewnetrzny_czujnik_CO2)
   END_RUNG wire#w3
   RUNG wire#w1
      { S7_Templates := "SrcType := Int" } GE_Contact(in1 := "Wejscia_PLC".Wewnetrzny_czujnik_CO2, in2 := 975)
      { S7_Templates := "SrcType := Int" } GT_Contact(in1 := "Wejscia_PLC".Wewnetrzny_czujnik_CO2, in2 := "Wejscia_PLC".Zewnetrzny_czujnik_CO2)
   END_RUNG wire#w4
   RUNG wire#powerrail
      Contact( #czy_manualny )
      I_Contact( #czy_automatyczny )
      Contact( "HMI".Otwarcie_okien_manual )
   END_RUNG wire#w4
   // the same network as SCL:
   "Siłownik_okien_otwieranie" := ((#czy_automatyczny AND NOT #czy_manualny AND (("HMI".System_okien_auto AND ("Wejscia_PLC".Czujnik_wiatru <= 35) AND (((#Histereza_plus < "HMI".Poziom_CO2_auto) AND ("Wejscia_PLC".Wewnetrzny_czujnik_CO2 > "Wejscia_PLC".Zewnetrzny_czujnik_CO2)) OR ((#Histereza_minus > "Wejscia_PLC".Wewnetrzny_czujnik_CO2) AND ("Wejscia_PLC".Wewnetrzny_czujnik_CO2 < "Wejscia_PLC".Zewnetrzny_czujnik_CO2))) AND (#Zakres_temp_dol <= "Wejscia_PLC".Temperatura_zewnetrzna) AND ("Wejscia_PLC".Temperatura_zewnetrzna <= #Zakres_temp_gora)) OR (("Wejscia_PLC".Wewnetrzny_czujnik_CO2 >= 975) AND ("Wejscia_PLC".Wewnetrzny_czujnik_CO2 > "Wejscia_PLC".Zewnetrzny_czujnik_CO2)))) OR (#czy_manualny AND NOT #czy_automatyczny AND "HMI".Otwarcie_okien_manual)) AND NOT "Siłownik_okien_zamykanie";
END_REGION

REGION Network 3: Warunki dla których okna są zamykane
   // W trybie automatycznym okna są zamykane: 1) gdy tryb okien został wyłączony przez użytkownika, 2) gdy stężenie CO2 w szklarni wynosi zadaną wartość tego parametru +- histereza, 3) gdy stężenie CO2 poza szklarnią jest mniejsze, niż wewnątrz, jeśli chcemy zwiększyć jego ilość oraz większe, gdy chcemy zmniejszyć jego ilość, 4) gdy tempperatura zewnętrzna różni się o ponad 5°C od zadanej, 5) gdy wiatr wieje z prędkością większą niż 35km/h, 6) gdy stężenie CO2 w szklarni nie przekracza 955ppm lub przekracza, ale stężenie CO2 poza szklarnią jest większe. W trybie manualnym okna są zamykane, gdy przełączk na HMI znajdzie się w pozycji "ZAMKNIĘTE".
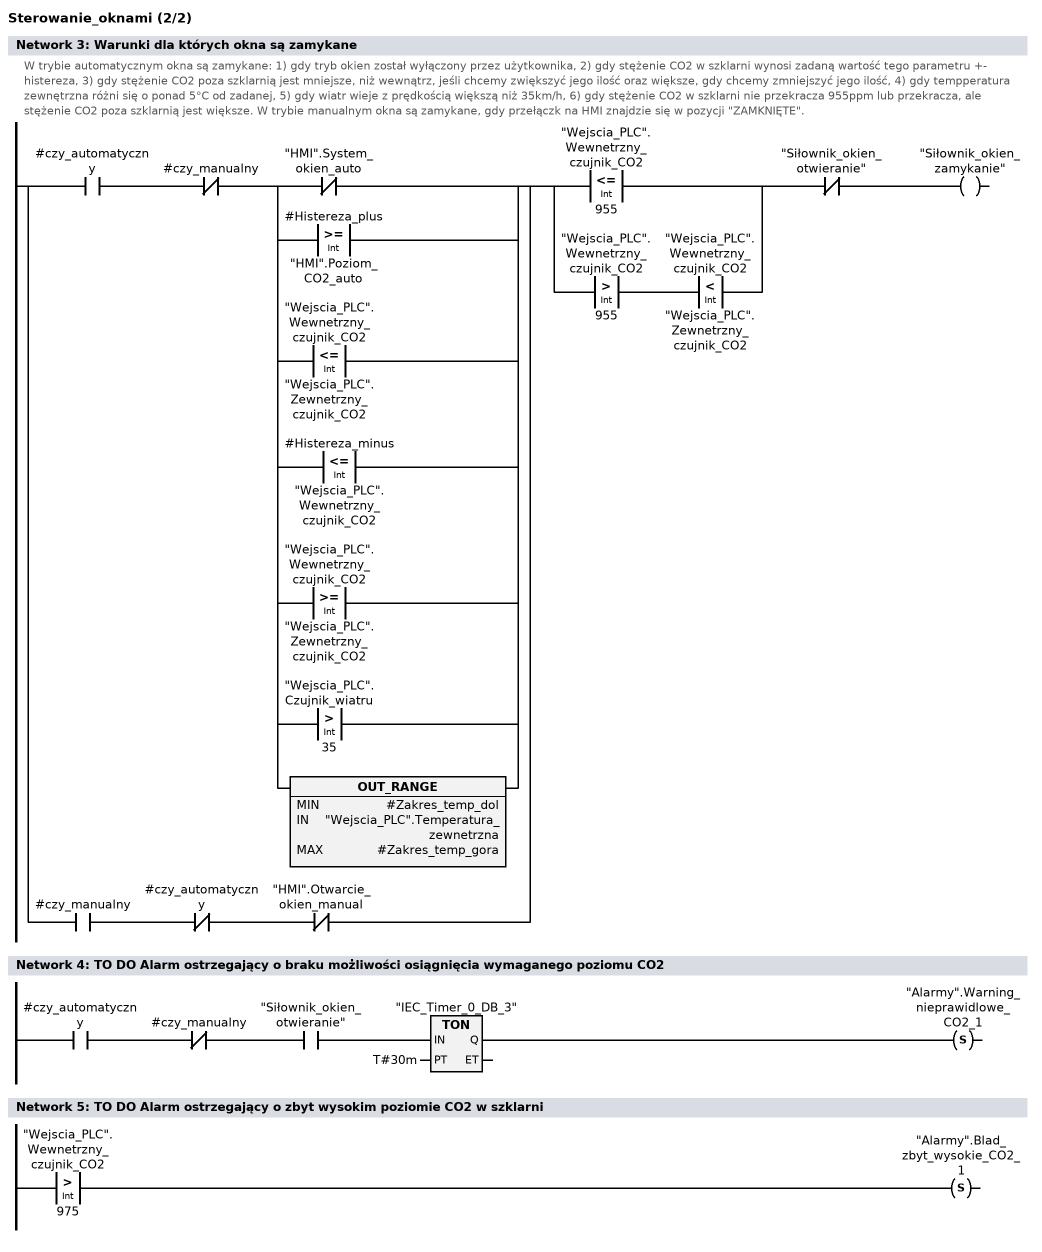
   "Siłownik_okien_zamykanie" := ((#czy_automatyczny AND NOT #czy_manualny AND (NOT "HMI".System_okien_auto OR (#Histereza_plus >= "HMI".Poziom_CO2_auto) OR ("Wejscia_PLC".Wewnetrzny_czujnik_CO2 <= "Wejscia_PLC".Zewnetrzny_czujnik_CO2) OR (#Histereza_minus <= "Wejscia_PLC".Wewnetrzny_czujnik_CO2) OR ("Wejscia_PLC".Wewnetrzny_czujnik_CO2 >= "Wejscia_PLC".Zewnetrzny_czujnik_CO2) OR ("Wejscia_PLC".Czujnik_wiatru > 35) OR ("Wejscia_PLC".Temperatura_zewnetrzna < #Zakres_temp_dol) OR ("Wejscia_PLC".Temperatura_zewnetrzna > #Zakres_temp_gora))) OR (#czy_manualny AND NOT #czy_automatyczny AND NOT "HMI".Otwarcie_okien_manual)) AND (("Wejscia_PLC".Wewnetrzny_czujnik_CO2 <= 955) OR (("Wejscia_PLC".Wewnetrzny_czujnik_CO2 > 955) AND ("Wejscia_PLC".Wewnetrzny_czujnik_CO2 < "Wejscia_PLC".Zewnetrzny_czujnik_CO2))) AND NOT "Siłownik_okien_otwieranie";
END_REGION

REGION Network 4: TO DO Alarm ostrzegający o braku możliwości osiągnięcia wymaganego poziomu CO2
   "IEC_Timer_0_DB_3".TON(IN := #czy_automatyczny AND NOT #czy_manualny AND "Siłownik_okien_otwieranie",
                          PT := T#30m);
   IF "IEC_Timer_0_DB_3".Q THEN "Alarmy".Warning_nieprawidlowe_CO2_1 := TRUE; END_IF;
END_REGION

REGION Network 5: TO DO Alarm ostrzegający o zbyt wysokim poziomie CO2 w szklarni
   RUNG wire#powerrail
      { S7_Templates := "SrcType := Int" } GT_Contact(in1 := "Wejscia_PLC".Wewnetrzny_czujnik_CO2, in2 := 975)
      S_Coil( "Alarmy".Blad_zbyt_wysokie_CO2_1 )
   END_RUNG
   // the same network as SCL:
   IF "Wejscia_PLC".Wewnetrzny_czujnik_CO2 > 975 THEN "Alarmy".Blad_zbyt_wysokie_CO2_1 := TRUE; END_IF;
END_REGION
END_FUNCTION

FUNCTION "SYMULACJA" : Void   // FC9, LAD
{ S7_Optimized_Access := 'TRUE' }
VERSION : 0.1
   VAR_INPUT
      counters : Bool;
   END_VAR
   VAR_TEMP
      temperatura_temp : Real;
      roznica_temperatur : Real;
      "wilgotność powietrza_temp" : Int;
      wilgotnosc_gleby_temp : Int;
      stezenie_CO2 : Int;
      natezenie_swiatla_temp : Int;
      odsloniecie_okna_temp : Real;
      pedkosc_wiatru_temp : Real;
      rand : Real;
      error : Bool;
      status : Int;
      sub_status : Int;
      rolety_temp : Real;
      test1 : Real;
   END_VAR
   VAR_TEMP   // added for the SCL form of the ladder/FBD networks
      _w1 : Bool;
   END_VAR
BEGIN

REGION Network 1: blok oblicza roznice temperatur
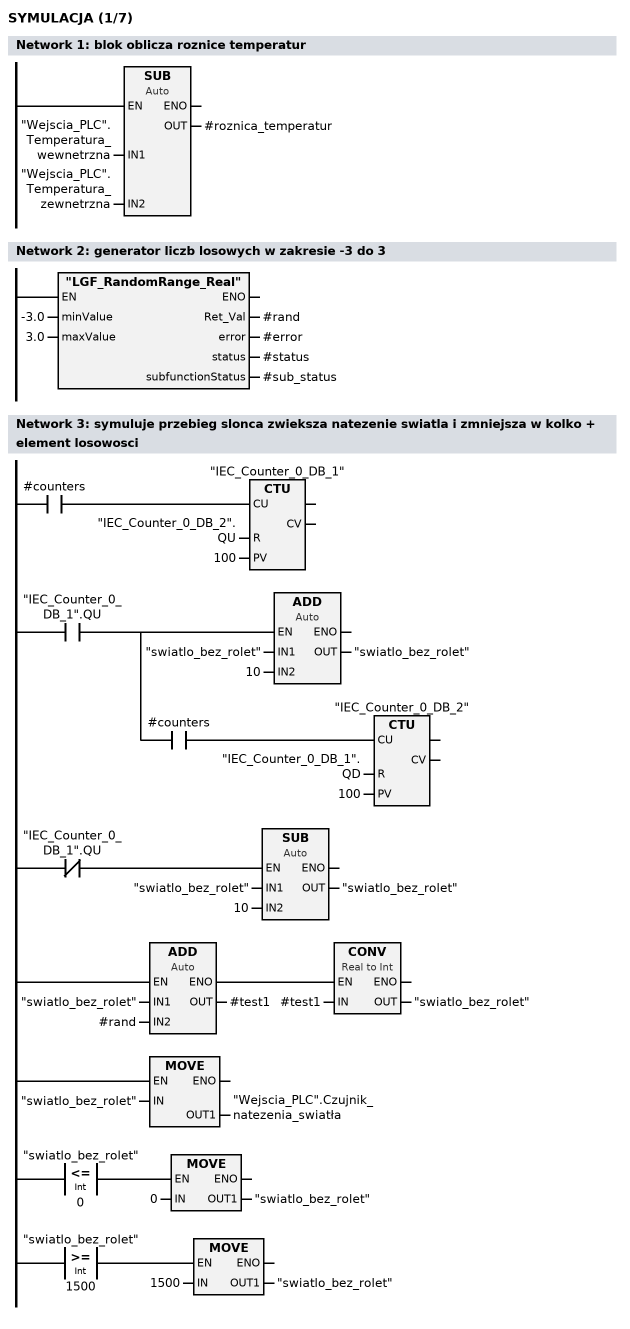
   RUNG wire#powerrail
      { S7_GenerateENO := "TRUE" } Sub(in1 := "Wejscia_PLC".Temperatura_wewnetrzna, in2 := "Wejscia_PLC".Temperatura_zewnetrzna, out => #roznica_temperatur)
   END_RUNG
   // the same network as SCL:
   #roznica_temperatur := "Wejscia_PLC".Temperatura_wewnetrzna - "Wejscia_PLC".Temperatura_zewnetrzna;
END_REGION

REGION Network 2: generator liczb losowych w zakresie -3 do 3
   RUNG wire#powerrail
      "LGF_RandomRange_Real"(minValue := -3.0, maxValue := 3.0, Ret_Val => #rand, error => #error, status => #status, subfunctionStatus => #sub_status)
   END_RUNG
   // the same network as SCL:
   #rand := "LGF_RandomRange_Real"(minValue := -3.0,
                           maxValue := 3.0,
                           error => #error,
                           status => #status,
                           subfunctionStatus => #sub_status);
END_REGION

REGION Network 3: symuluje przebieg slonca zwieksza natezenie swiatla i zmniejsza w kolko + element losowosci
   // ENO of a box is taken as its EN; it also drops when the box reports an error
   "IEC_Counter_0_DB_1".CTU(CU := #counters, R := "IEC_Counter_0_DB_2".QU, PV := 100);
   IF "IEC_Counter_0_DB_1".QU THEN "swiatlo_bez_rolet" := "swiatlo_bez_rolet" + 10; END_IF;
   "IEC_Counter_0_DB_2".CTU(CU := "IEC_Counter_0_DB_1".QU AND #counters,
                           R := "IEC_Counter_0_DB_1".QD,
                           PV := 100);
   IF NOT "IEC_Counter_0_DB_1".QU THEN "swiatlo_bez_rolet" := "swiatlo_bez_rolet" - 10; END_IF;
   #test1 := "swiatlo_bez_rolet" + #rand;
   "swiatlo_bez_rolet" := REAL_TO_INT(#test1);
   "Wejscia_PLC".Czujnik_natezenia_swiatła := "swiatlo_bez_rolet";
   IF "swiatlo_bez_rolet" <= 0 THEN "swiatlo_bez_rolet" := 0; END_IF;
   IF "swiatlo_bez_rolet" >= 1500 THEN "swiatlo_bez_rolet" := 1500; END_IF;
END_REGION

REGION Network 4: funkcja oblicza liniową zależność natężenia światła od zasłonięcia rolet
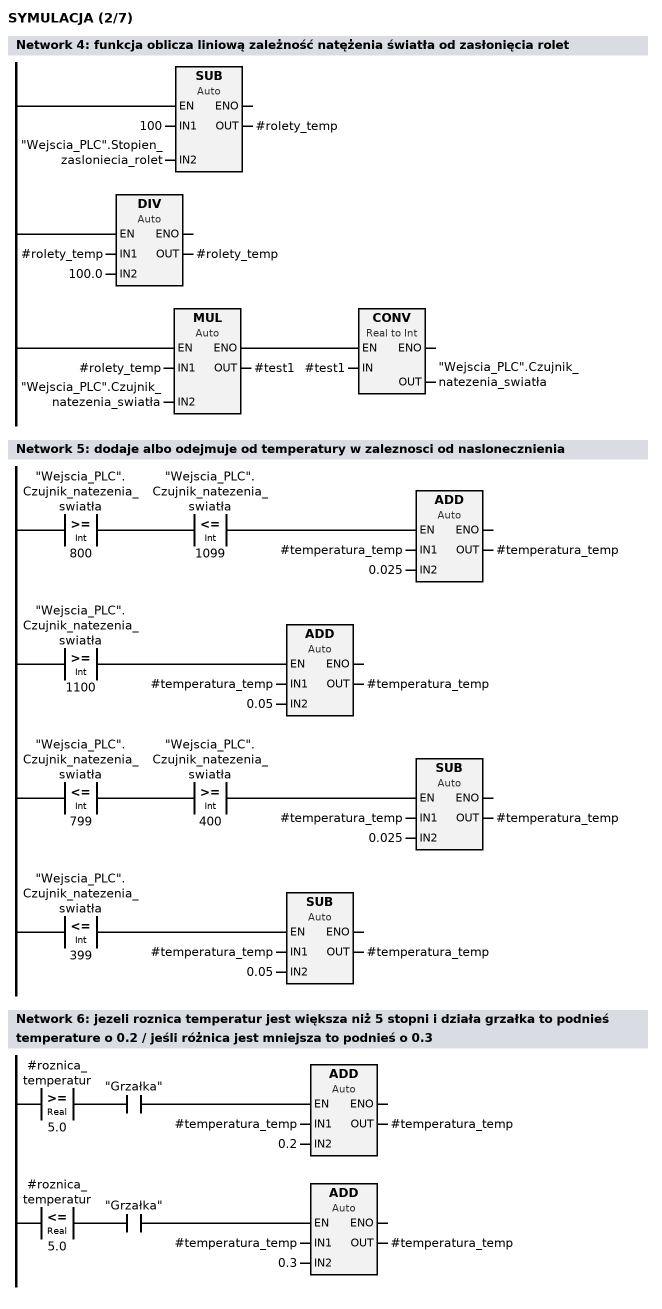
   RUNG wire#powerrail
      { S7_GenerateENO := "TRUE" } Sub(in1 := 100, in2 := "Wejscia_PLC".Stopien_zasloniecia_rolet, out => #rolety_temp)
   END_RUNG
   RUNG wire#powerrail
      { S7_GenerateENO := "TRUE" } Div(in1 := #rolety_temp, in2 := 100.0, out => #rolety_temp)
   END_RUNG
   RUNG wire#powerrail
      { S7_GenerateENO := "TRUE" } Mul(in1 := #rolety_temp, in2 := "Wejscia_PLC".Czujnik_natezenia_swiatła, out => #test1)
      { S7_Templates := "[SrcType := Real, DestType := Int]"; S7_GenerateENO := "TRUE" } Convert(in := #test1, out => "Wejscia_PLC".Czujnik_natezenia_swiatła)
   END_RUNG
   // the same network as SCL:
   // ENO of a box is taken as its EN; it also drops when the box reports an error
   #rolety_temp := 100 - "Wejscia_PLC".Stopien_zasloniecia_rolet;
   #rolety_temp := #rolety_temp / 100.0;
   #test1 := #rolety_temp * "Wejscia_PLC".Czujnik_natezenia_swiatła;
   "Wejscia_PLC".Czujnik_natezenia_swiatła := REAL_TO_INT(#test1);
END_REGION

REGION Network 5: dodaje albo odejmuje od temperatury w zaleznosci od naslonecznienia
   RUNG wire#powerrail
      { S7_Templates := "SrcType := Int" } GE_Contact(in1 := "Wejscia_PLC".Czujnik_natezenia_swiatła, in2 := 800)
      { S7_Templates := "SrcType := Int" } LE_Contact(in1 := "Wejscia_PLC".Czujnik_natezenia_swiatła, in2 := 1099)
      { S7_GenerateENO := "TRUE" } Add(in1 := #temperatura_temp, in2 := 0.025, out => #temperatura_temp)
   END_RUNG
   RUNG wire#powerrail
      { S7_Templates := "SrcType := Int" } GE_Contact(in1 := "Wejscia_PLC".Czujnik_natezenia_swiatła, in2 := 1100)
      { S7_GenerateENO := "TRUE" } Add(in1 := #temperatura_temp, in2 := 0.05, out => #temperatura_temp)
   END_RUNG
   RUNG wire#powerrail
      { S7_Templates := "SrcType := Int" } LE_Contact(in1 := "Wejscia_PLC".Czujnik_natezenia_swiatła, in2 := 799)
      { S7_Templates := "SrcType := Int" } GE_Contact(in1 := "Wejscia_PLC".Czujnik_natezenia_swiatła, in2 := 400)
      { S7_GenerateENO := "TRUE" } Sub(in1 := #temperatura_temp, in2 := 0.025, out => #temperatura_temp)
   END_RUNG
   RUNG wire#powerrail
      { S7_Templates := "SrcType := Int" } LE_Contact(in1 := "Wejscia_PLC".Czujnik_natezenia_swiatła, in2 := 399)
      { S7_GenerateENO := "TRUE" } Sub(in1 := #temperatura_temp, in2 := 0.05, out => #temperatura_temp)
   END_RUNG
   // the same network as SCL:
   IF ("Wejscia_PLC".Czujnik_natezenia_swiatła >= 800) AND ("Wejscia_PLC".Czujnik_natezenia_swiatła <= 1099) THEN
       #temperatura_temp := #temperatura_temp + 0.025;
   END_IF;
   IF "Wejscia_PLC".Czujnik_natezenia_swiatła >= 1100 THEN
       #temperatura_temp := #temperatura_temp + 0.05;
   END_IF;
   IF ("Wejscia_PLC".Czujnik_natezenia_swiatła <= 799) AND ("Wejscia_PLC".Czujnik_natezenia_swiatła >= 400) THEN
       #temperatura_temp := #temperatura_temp - 0.025;
   END_IF;
   IF "Wejscia_PLC".Czujnik_natezenia_swiatła <= 399 THEN
       #temperatura_temp := #temperatura_temp - 0.05;
   END_IF;
END_REGION

REGION Network 6: jezeli roznica temperatur jest większa niż 5 stopni i działa grzałka to podnieś temperature o 0.2 / jeśli różnica jest mniejsza to podnieś o 0.3
   RUNG wire#powerrail
      { S7_Templates := "SrcType := Real" } GE_Contact(in1 := #roznica_temperatur, in2 := 5.0)
      Contact( "Grzałka" )
      { S7_GenerateENO := "TRUE" } Add(in1 := #temperatura_temp, in2 := 0.2, out => #temperatura_temp)
   END_RUNG
   RUNG wire#powerrail
      { S7_Templates := "SrcType := Real" } LE_Contact(in1 := #roznica_temperatur, in2 := 5.0)
      Contact( "Grzałka" )
      { S7_GenerateENO := "TRUE" } Add(in1 := #temperatura_temp, in2 := 0.3, out => #temperatura_temp)
   END_RUNG
   // the same network as SCL:
   IF (#roznica_temperatur >= 5.0) AND "Grzałka" THEN #temperatura_temp := #temperatura_temp + 0.2; END_IF;
   IF (#roznica_temperatur <= 5.0) AND "Grzałka" THEN #temperatura_temp := #temperatura_temp + 0.3; END_IF;
END_REGION

REGION Network 7: jezeli działa wentylator to obniż temperature o 0.1
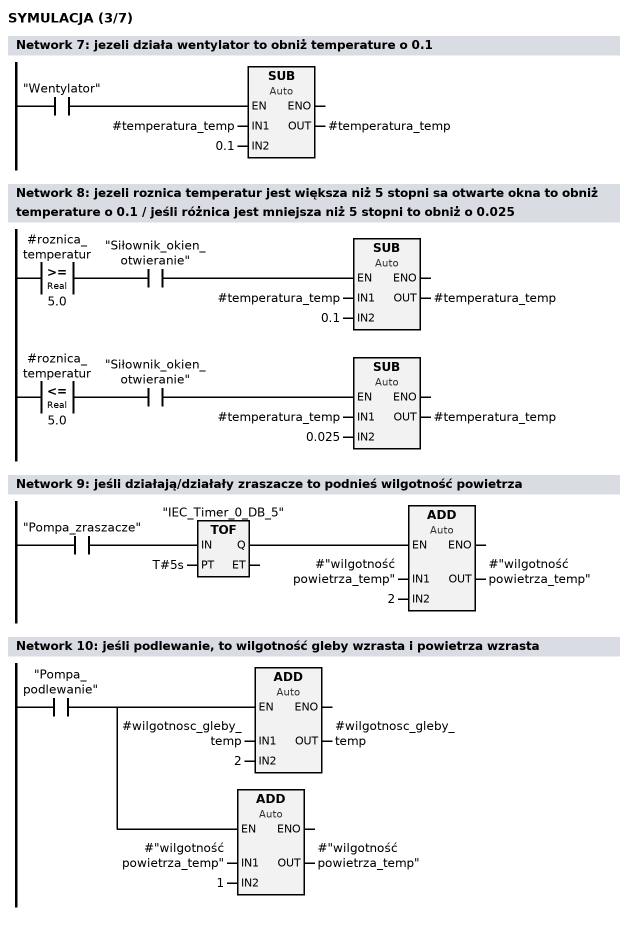
   RUNG wire#powerrail
      Contact( "Wentylator" )
      { S7_GenerateENO := "TRUE" } Sub(in1 := #temperatura_temp, in2 := 0.1, out => #temperatura_temp)
   END_RUNG
   // the same network as SCL:
   IF "Wentylator" THEN #temperatura_temp := #temperatura_temp - 0.1; END_IF;
END_REGION

REGION Network 8: jezeli roznica temperatur jest większa niż 5 stopni sa otwarte okna to obniż temperature o 0.1 / jeśli różnica jest mniejsza niż 5 stopni to obniż o 0.025
   RUNG wire#powerrail
      { S7_Templates := "SrcType := Real" } GE_Contact(in1 := #roznica_temperatur, in2 := 5.0)
      Contact( "Siłownik_okien_otwieranie" )
      { S7_GenerateENO := "TRUE" } Sub(in1 := #temperatura_temp, in2 := 0.1, out => #temperatura_temp)
   END_RUNG
   RUNG wire#powerrail
      { S7_Templates := "SrcType := Real" } LE_Contact(in1 := #roznica_temperatur, in2 := 5.0)
      Contact( "Siłownik_okien_otwieranie" )
      { S7_GenerateENO := "TRUE" } Sub(in1 := #temperatura_temp, in2 := 0.025, out => #temperatura_temp)
   END_RUNG
   // the same network as SCL:
   IF (#roznica_temperatur >= 5.0) AND "Siłownik_okien_otwieranie" THEN
       #temperatura_temp := #temperatura_temp - 0.1;
   END_IF;
   IF (#roznica_temperatur <= 5.0) AND "Siłownik_okien_otwieranie" THEN
       #temperatura_temp := #temperatura_temp - 0.025;
   END_IF;
END_REGION

REGION Network 9: jeśli działają/działały zraszacze to podnieś wilgotność powietrza
   "IEC_Timer_0_DB_5".TOF(IN := "Pompa_zraszacze", PT := T#5s);
   IF "IEC_Timer_0_DB_5".Q THEN #"wilgotność powietrza_temp" := #"wilgotność powietrza_temp" + 2; END_IF;
END_REGION

REGION Network 10: jeśli podlewanie, to wilgotność gleby wzrasta i powietrza wzrasta
   RUNG wire#powerrail
      Contact( "Pompa_podlewanie" )
      wire#w1
      { S7_GenerateENO := "TRUE" } Add(in1 := #wilgotnosc_gleby_temp, in2 := 2, out => #wilgotnosc_gleby_temp)
   END_RUNG
   RUNG wire#w1
      { S7_GenerateENO := "TRUE" } Add(in1 := #"wilgotność powietrza_temp", in2 := 1, out => #"wilgotność powietrza_temp")
   END_RUNG
   // the same network as SCL:
   IF "Pompa_podlewanie" THEN
       #wilgotnosc_gleby_temp := #wilgotnosc_gleby_temp + 2;
       #"wilgotność powietrza_temp" := #"wilgotność powietrza_temp" + 1;
   END_IF;
END_REGION

REGION Network 11: realizacja zaleznosci odslaniania i zaslaniania rolet, od stopnia zasłonięcia
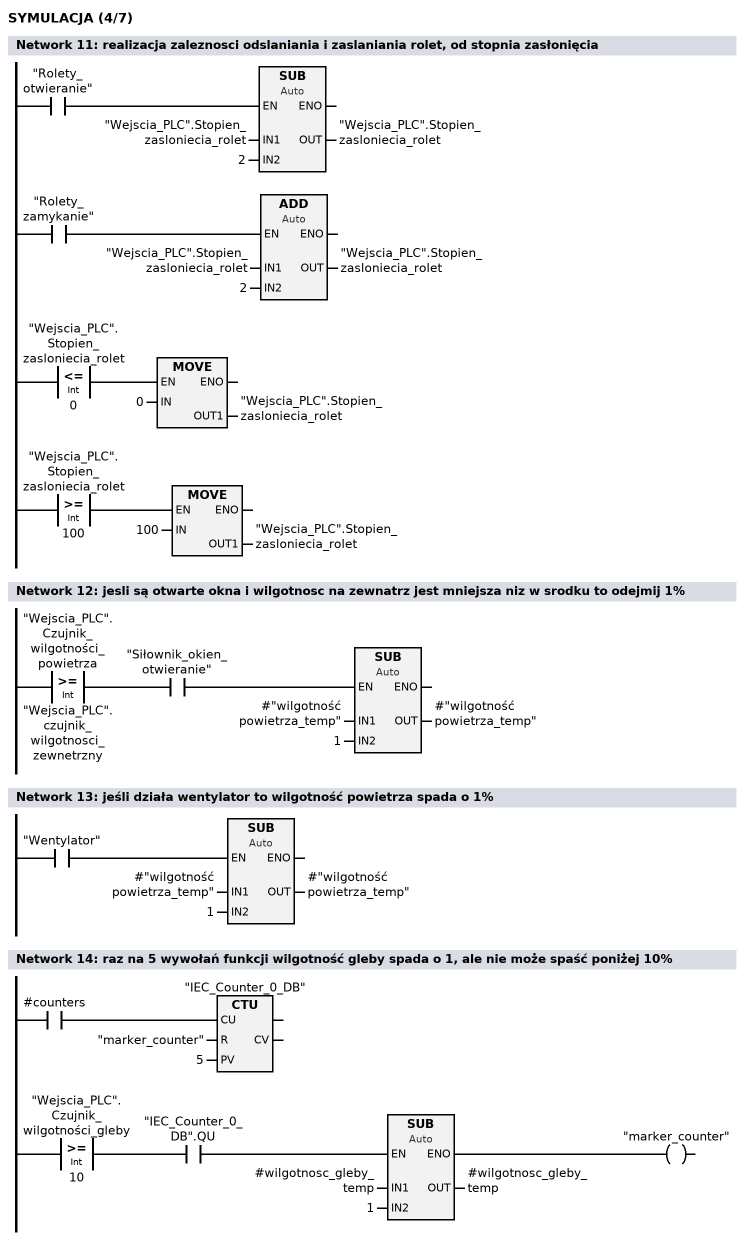
   RUNG wire#powerrail
      Contact( "Rolety_otwieranie" )
      { S7_GenerateENO := "TRUE" } Sub(in1 := "Wejscia_PLC".Stopien_zasloniecia_rolet, in2 := 2, out => "Wejscia_PLC".Stopien_zasloniecia_rolet)
   END_RUNG
   RUNG wire#powerrail
      Contact( "Rolety_zamykanie" )
      { S7_GenerateENO := "TRUE" } Add(in1 := "Wejscia_PLC".Stopien_zasloniecia_rolet, in2 := 2, out => "Wejscia_PLC".Stopien_zasloniecia_rolet)
   END_RUNG
   RUNG wire#powerrail
      { S7_Templates := "SrcType := Int" } LE_Contact(in1 := "Wejscia_PLC".Stopien_zasloniecia_rolet, in2 := 0)
      { S7_GenerateENO := "TRUE" } Move(in := 0, out1 => "Wejscia_PLC".Stopien_zasloniecia_rolet)
   END_RUNG
   RUNG wire#powerrail
      { S7_Templates := "SrcType := Int" } GE_Contact(in1 := "Wejscia_PLC".Stopien_zasloniecia_rolet, in2 := 100)
      { S7_GenerateENO := "TRUE" } Move(in := 100, out1 => "Wejscia_PLC".Stopien_zasloniecia_rolet)
   END_RUNG
   // the same network as SCL:
   IF "Rolety_otwieranie" THEN
       "Wejscia_PLC".Stopien_zasloniecia_rolet := "Wejscia_PLC".Stopien_zasloniecia_rolet - 2;
   END_IF;
   IF "Rolety_zamykanie" THEN
       "Wejscia_PLC".Stopien_zasloniecia_rolet := "Wejscia_PLC".Stopien_zasloniecia_rolet + 2;
   END_IF;
   IF "Wejscia_PLC".Stopien_zasloniecia_rolet <= 0 THEN "Wejscia_PLC".Stopien_zasloniecia_rolet := 0; END_IF;
   IF "Wejscia_PLC".Stopien_zasloniecia_rolet >= 100 THEN
       "Wejscia_PLC".Stopien_zasloniecia_rolet := 100;
   END_IF;
END_REGION

REGION Network 12: jesli są otwarte okna i wilgotnosc na zewnatrz jest mniejsza niz w srodku to odejmij 1%
   RUNG wire#powerrail
      { S7_Templates := "SrcType := Int" } GE_Contact(in1 := "Wejscia_PLC".Czujnik_wilgotności_powietrza, in2 := "Wejscia_PLC".czujnik_wilgotnosci_zewnetrzny)
      Contact( "Siłownik_okien_otwieranie" )
      { S7_GenerateENO := "TRUE" } Sub(in1 := #"wilgotność powietrza_temp", in2 := 1, out => #"wilgotność powietrza_temp")
   END_RUNG
   // the same network as SCL:
   IF ("Wejscia_PLC".Czujnik_wilgotności_powietrza >= "Wejscia_PLC".czujnik_wilgotnosci_zewnetrzny) AND "Siłownik_okien_otwieranie" THEN
       #"wilgotność powietrza_temp" := #"wilgotność powietrza_temp" - 1;
   END_IF;
END_REGION

REGION Network 13: jeśli działa wentylator to wilgotność powietrza spada o 1%
   RUNG wire#powerrail
      Contact( "Wentylator" )
      { S7_GenerateENO := "TRUE" } Sub(in1 := #"wilgotność powietrza_temp", in2 := 1, out => #"wilgotność powietrza_temp")
   END_RUNG
   // the same network as SCL:
   IF "Wentylator" THEN #"wilgotność powietrza_temp" := #"wilgotność powietrza_temp" - 1; END_IF;
END_REGION

REGION Network 14: raz na 5 wywołań funkcji wilgotność gleby spada o 1, ale nie może spaść poniżej 10%
   // ENO of a box is taken as its EN; it also drops when the box reports an error
   "IEC_Counter_0_DB".CTU(CU := #counters, R := "marker_counter", PV := 5);
   #_w1 := ("Wejscia_PLC".Czujnik_wilgotności_gleby >= 10) AND "IEC_Counter_0_DB".QU;
   IF #_w1 THEN #wilgotnosc_gleby_temp := #wilgotnosc_gleby_temp - 1; END_IF;
   "marker_counter" := #_w1;
END_REGION

REGION Network 15: jeśli stężenie na zewnątrz jest mniejsze, a są otwarte okna to zmniejsz stężenie CO2
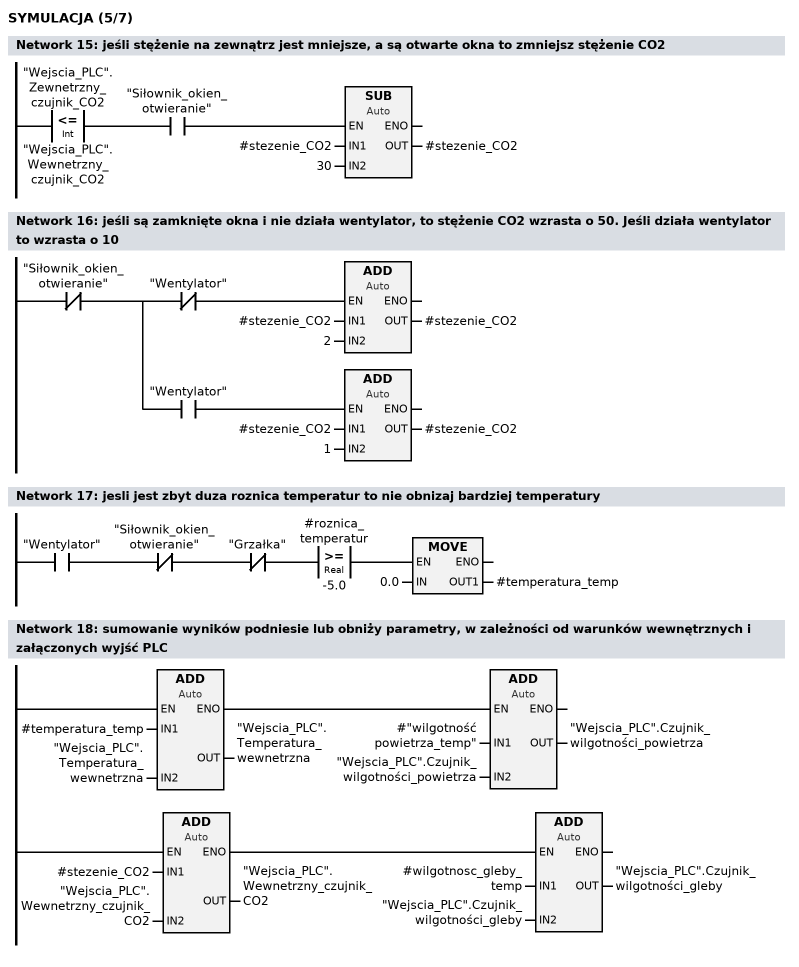
   RUNG wire#powerrail
      { S7_Templates := "SrcType := Int" } LE_Contact(in1 := "Wejscia_PLC".Zewnetrzny_czujnik_CO2, in2 := "Wejscia_PLC".Wewnetrzny_czujnik_CO2)
      Contact( "Siłownik_okien_otwieranie" )
      { S7_GenerateENO := "TRUE" } Sub(in1 := #stezenie_CO2, in2 := 30, out => #stezenie_CO2)
   END_RUNG
   // the same network as SCL:
   IF ("Wejscia_PLC".Zewnetrzny_czujnik_CO2 <= "Wejscia_PLC".Wewnetrzny_czujnik_CO2) AND "Siłownik_okien_otwieranie" THEN
       #stezenie_CO2 := #stezenie_CO2 - 30;
   END_IF;
END_REGION

REGION Network 16: jeśli są zamknięte okna i nie działa wentylator, to stężenie CO2 wzrasta o 50. Jeśli działa wentylator to wzrasta o 10
   RUNG wire#powerrail
      I_Contact( "Siłownik_okien_otwieranie" )
      wire#w1
      I_Contact( "Wentylator" )
      { S7_GenerateENO := "TRUE" } Add(in1 := #stezenie_CO2, in2 := 2, out => #stezenie_CO2)
   END_RUNG
   RUNG wire#w1
      Contact( "Wentylator" )
      { S7_GenerateENO := "TRUE" } Add(in1 := #stezenie_CO2, in2 := 1, out => #stezenie_CO2)
   END_RUNG
   // the same network as SCL:
   #_w1 := NOT "Siłownik_okien_otwieranie";
   IF #_w1 AND NOT "Wentylator" THEN #stezenie_CO2 := #stezenie_CO2 + 2; END_IF;
   IF #_w1 AND "Wentylator" THEN #stezenie_CO2 := #stezenie_CO2 + 1; END_IF;
END_REGION

REGION Network 17: jesli jest zbyt duza roznica temperatur to nie obnizaj bardziej temperatury
   RUNG wire#powerrail
      Contact( "Wentylator" )
      I_Contact( "Siłownik_okien_otwieranie" )
      I_Contact( "Grzałka" )
      { S7_Templates := "SrcType := Real" } GE_Contact(in1 := #roznica_temperatur, in2 := -5.0)
      { S7_GenerateENO := "TRUE" } Move(in := 0.0, out1 => #temperatura_temp)
   END_RUNG
   // the same network as SCL:
   IF "Wentylator" AND NOT "Siłownik_okien_otwieranie" AND NOT "Grzałka" AND (#roznica_temperatur >= (-5.0)) THEN
       #temperatura_temp := 0.0;
   END_IF;
END_REGION

REGION Network 18: sumowanie wyników podniesie lub obniży parametry, w zależności od warunków wewnętrznych i załączonych wyjść PLC
   RUNG wire#powerrail
      { S7_GenerateENO := "TRUE" } Add(in1 := #temperatura_temp, in2 := "Wejscia_PLC".Temperatura_wewnetrzna, out => "Wejscia_PLC".Temperatura_wewnetrzna)
      { S7_GenerateENO := "TRUE" } Add(in1 := #"wilgotność powietrza_temp", in2 := "Wejscia_PLC".Czujnik_wilgotności_powietrza, out => "Wejscia_PLC".Czujnik_wilgotności_powietrza)
   END_RUNG
   RUNG wire#powerrail
      { S7_GenerateENO := "TRUE" } Add(in1 := #stezenie_CO2, in2 := "Wejscia_PLC".Wewnetrzny_czujnik_CO2, out => "Wejscia_PLC".Wewnetrzny_czujnik_CO2)
      { S7_GenerateENO := "TRUE" } Add(in1 := #wilgotnosc_gleby_temp, in2 := "Wejscia_PLC".Czujnik_wilgotności_gleby, out => "Wejscia_PLC".Czujnik_wilgotności_gleby)
   END_RUNG
   // the same network as SCL:
   // ENO of a box is taken as its EN; it also drops when the box reports an error
   "Wejscia_PLC".Temperatura_wewnetrzna := #temperatura_temp + "Wejscia_PLC".Temperatura_wewnetrzna;
   "Wejscia_PLC".Czujnik_wilgotności_powietrza := #"wilgotność powietrza_temp" + "Wejscia_PLC".Czujnik_wilgotności_powietrza;
   "Wejscia_PLC".Wewnetrzny_czujnik_CO2 := #stezenie_CO2 + "Wejscia_PLC".Wewnetrzny_czujnik_CO2;
   "Wejscia_PLC".Czujnik_wilgotności_gleby := #wilgotnosc_gleby_temp + "Wejscia_PLC".Czujnik_wilgotności_gleby;
END_REGION

REGION Network 19: zabezpieczenie, przed przekroczeniem wartości krytycznych czujników + zabezpieczenia fizyczne np. procenty tylko w zakresie(0-100)
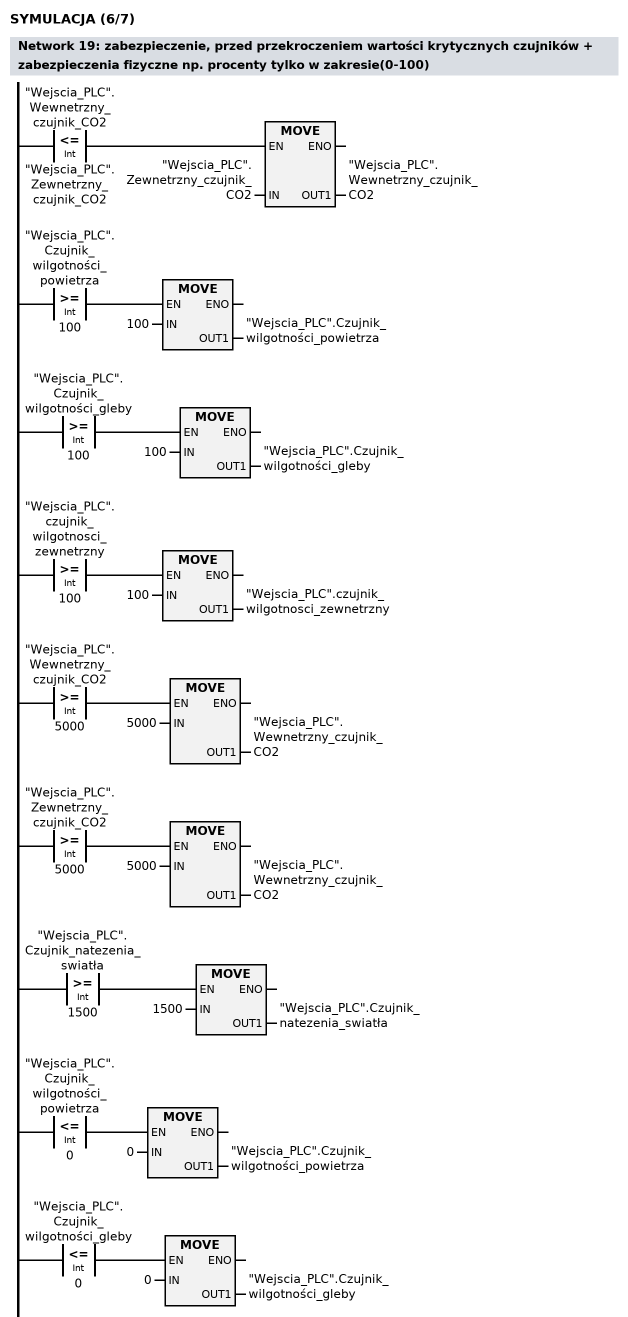
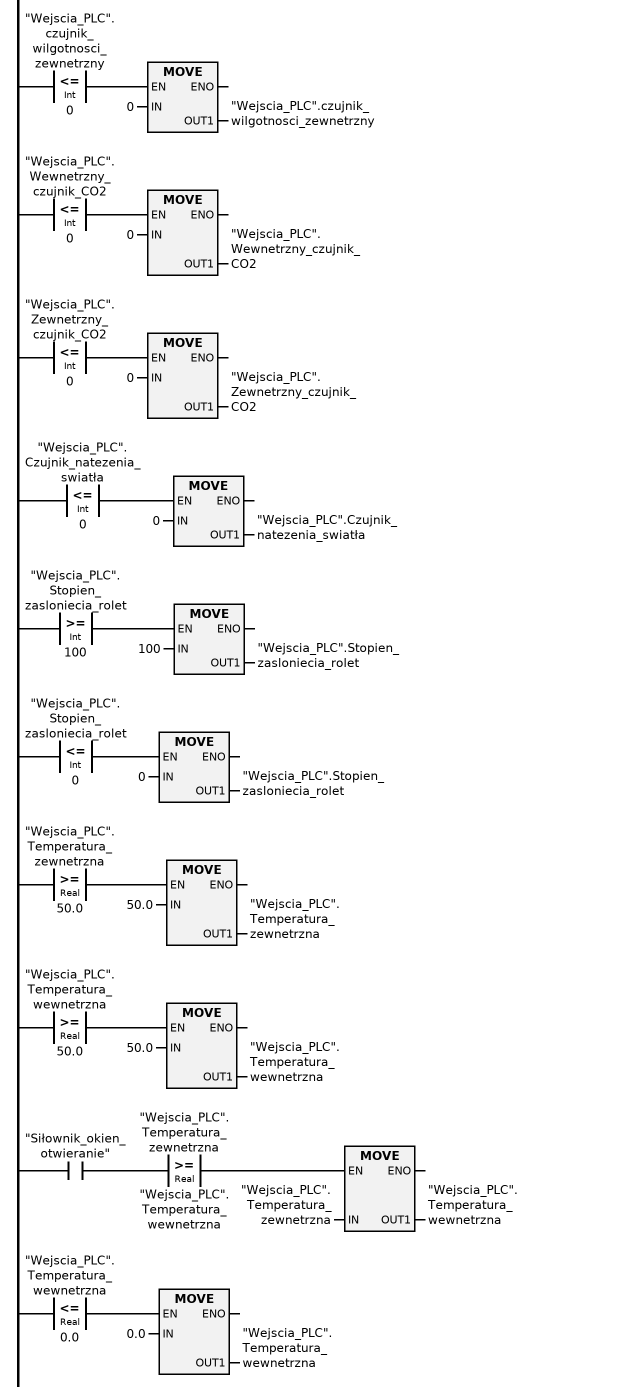
   RUNG wire#powerrail
      { S7_Templates := "SrcType := Int" } LE_Contact(in1 := "Wejscia_PLC".Wewnetrzny_czujnik_CO2, in2 := "Wejscia_PLC".Zewnetrzny_czujnik_CO2)
      { S7_GenerateENO := "TRUE" } Move(in := "Wejscia_PLC".Zewnetrzny_czujnik_CO2, out1 => "Wejscia_PLC".Wewnetrzny_czujnik_CO2)
   END_RUNG
   RUNG wire#powerrail
      { S7_Templates := "SrcType := Int" } GE_Contact(in1 := "Wejscia_PLC".Czujnik_wilgotności_powietrza, in2 := 100)
      { S7_GenerateENO := "TRUE" } Move(in := 100, out1 => "Wejscia_PLC".Czujnik_wilgotności_powietrza)
   END_RUNG
   RUNG wire#powerrail
      { S7_Templates := "SrcType := Int" } GE_Contact(in1 := "Wejscia_PLC".Czujnik_wilgotności_gleby, in2 := 100)
      { S7_GenerateENO := "TRUE" } Move(in := 100, out1 => "Wejscia_PLC".Czujnik_wilgotności_gleby)
   END_RUNG
   RUNG wire#powerrail
      { S7_Templates := "SrcType := Int" } GE_Contact(in1 := "Wejscia_PLC".czujnik_wilgotnosci_zewnetrzny, in2 := 100)
      { S7_GenerateENO := "TRUE" } Move(in := 100, out1 => "Wejscia_PLC".czujnik_wilgotnosci_zewnetrzny)
   END_RUNG
   RUNG wire#powerrail
      { S7_Templates := "SrcType := Int" } GE_Contact(in1 := "Wejscia_PLC".Wewnetrzny_czujnik_CO2, in2 := 5000)
      { S7_GenerateENO := "TRUE" } Move(in := 5000, out1 => "Wejscia_PLC".Wewnetrzny_czujnik_CO2)
   END_RUNG
   RUNG wire#powerrail
      { S7_Templates := "SrcType := Int" } GE_Contact(in1 := "Wejscia_PLC".Zewnetrzny_czujnik_CO2, in2 := 5000)
      { S7_GenerateENO := "TRUE" } Move(in := 5000, out1 => "Wejscia_PLC".Wewnetrzny_czujnik_CO2)
   END_RUNG
   RUNG wire#powerrail
      { S7_Templates := "SrcType := Int" } GE_Contact(in1 := "Wejscia_PLC".Czujnik_natezenia_swiatła, in2 := 1500)
      { S7_GenerateENO := "TRUE" } Move(in := 1500, out1 => "Wejscia_PLC".Czujnik_natezenia_swiatła)
   END_RUNG
   RUNG wire#powerrail
      { S7_Templates := "SrcType := Int" } LE_Contact(in1 := "Wejscia_PLC".Czujnik_wilgotności_powietrza, in2 := 0)
      { S7_GenerateENO := "TRUE" } Move(in := 0, out1 => "Wejscia_PLC".Czujnik_wilgotności_powietrza)
   END_RUNG
   RUNG wire#powerrail
      { S7_Templates := "SrcType := Int" } LE_Contact(in1 := "Wejscia_PLC".Czujnik_wilgotności_gleby, in2 := 0)
      { S7_GenerateENO := "TRUE" } Move(in := 0, out1 => "Wejscia_PLC".Czujnik_wilgotności_gleby)
   END_RUNG
   RUNG wire#powerrail
      { S7_Templates := "SrcType := Int" } LE_Contact(in1 := "Wejscia_PLC".czujnik_wilgotnosci_zewnetrzny, in2 := 0)
      { S7_GenerateENO := "TRUE" } Move(in := 0, out1 => "Wejscia_PLC".czujnik_wilgotnosci_zewnetrzny)
   END_RUNG
   RUNG wire#powerrail
      { S7_Templates := "SrcType := Int" } LE_Contact(in1 := "Wejscia_PLC".Wewnetrzny_czujnik_CO2, in2 := 0)
      { S7_GenerateENO := "TRUE" } Move(in := 0, out1 => "Wejscia_PLC".Wewnetrzny_czujnik_CO2)
   END_RUNG
   RUNG wire#powerrail
      { S7_Templates := "SrcType := Int" } LE_Contact(in1 := "Wejscia_PLC".Zewnetrzny_czujnik_CO2, in2 := 0)
      { S7_GenerateENO := "TRUE" } Move(in := 0, out1 => "Wejscia_PLC".Zewnetrzny_czujnik_CO2)
   END_RUNG
   RUNG wire#powerrail
      { S7_Templates := "SrcType := Int" } LE_Contact(in1 := "Wejscia_PLC".Czujnik_natezenia_swiatła, in2 := 0)
      { S7_GenerateENO := "TRUE" } Move(in := 0, out1 => "Wejscia_PLC".Czujnik_natezenia_swiatła)
   END_RUNG
   RUNG wire#powerrail
      { S7_Templates := "SrcType := Int" } GE_Contact(in1 := "Wejscia_PLC".Stopien_zasloniecia_rolet, in2 := 100)
      { S7_GenerateENO := "TRUE" } Move(in := 100, out1 => "Wejscia_PLC".Stopien_zasloniecia_rolet)
   END_RUNG
   RUNG wire#powerrail
      { S7_Templates := "SrcType := Int" } LE_Contact(in1 := "Wejscia_PLC".Stopien_zasloniecia_rolet, in2 := 0)
      { S7_GenerateENO := "TRUE" } Move(in := 0, out1 => "Wejscia_PLC".Stopien_zasloniecia_rolet)
   END_RUNG
   RUNG wire#powerrail
      { S7_Templates := "SrcType := Real" } GE_Contact(in1 := "Wejscia_PLC".Temperatura_zewnetrzna, in2 := 50.0)
      { S7_GenerateENO := "TRUE" } Move(in := 50.0, out1 => "Wejscia_PLC".Temperatura_zewnetrzna)
   END_RUNG
   RUNG wire#powerrail
      { S7_Templates := "SrcType := Real" } GE_Contact(in1 := "Wejscia_PLC".Temperatura_wewnetrzna, in2 := 50.0)
      { S7_GenerateENO := "TRUE" } Move(in := 50.0, out1 => "Wejscia_PLC".Temperatura_wewnetrzna)
   END_RUNG
   RUNG wire#powerrail
      Contact( "Siłownik_okien_otwieranie" )
      { S7_Templates := "SrcType := Real" } GE_Contact(in1 := "Wejscia_PLC".Temperatura_zewnetrzna, in2 := "Wejscia_PLC".Temperatura_wewnetrzna)
      { S7_GenerateENO := "TRUE" } Move(in := "Wejscia_PLC".Temperatura_zewnetrzna, out1 => "Wejscia_PLC".Temperatura_wewnetrzna)
   END_RUNG
   RUNG wire#powerrail
      { S7_Templates := "SrcType := Real" } LE_Contact(in1 := "Wejscia_PLC".Temperatura_wewnetrzna, in2 := 0.0)
      { S7_GenerateENO := "TRUE" } Move(in := 0.0, out1 => "Wejscia_PLC".Temperatura_wewnetrzna)
   END_RUNG
   // the same network as SCL:
   IF "Wejscia_PLC".Wewnetrzny_czujnik_CO2 <= "Wejscia_PLC".Zewnetrzny_czujnik_CO2 THEN
       "Wejscia_PLC".Wewnetrzny_czujnik_CO2 := "Wejscia_PLC".Zewnetrzny_czujnik_CO2;
   END_IF;
   IF "Wejscia_PLC".Czujnik_wilgotności_powietrza >= 100 THEN
       "Wejscia_PLC".Czujnik_wilgotności_powietrza := 100;
   END_IF;
   IF "Wejscia_PLC".Czujnik_wilgotności_gleby >= 100 THEN
       "Wejscia_PLC".Czujnik_wilgotności_gleby := 100;
   END_IF;
   IF "Wejscia_PLC".czujnik_wilgotnosci_zewnetrzny >= 100 THEN
       "Wejscia_PLC".czujnik_wilgotnosci_zewnetrzny := 100;
   END_IF;
   IF "Wejscia_PLC".Wewnetrzny_czujnik_CO2 >= 5000 THEN "Wejscia_PLC".Wewnetrzny_czujnik_CO2 := 5000; END_IF;
   IF "Wejscia_PLC".Zewnetrzny_czujnik_CO2 >= 5000 THEN "Wejscia_PLC".Wewnetrzny_czujnik_CO2 := 5000; END_IF;
   IF "Wejscia_PLC".Czujnik_natezenia_swiatła >= 1500 THEN
       "Wejscia_PLC".Czujnik_natezenia_swiatła := 1500;
   END_IF;
   IF "Wejscia_PLC".Czujnik_wilgotności_powietrza <= 0 THEN
       "Wejscia_PLC".Czujnik_wilgotności_powietrza := 0;
   END_IF;
   IF "Wejscia_PLC".Czujnik_wilgotności_gleby <= 0 THEN "Wejscia_PLC".Czujnik_wilgotności_gleby := 0; END_IF;
   IF "Wejscia_PLC".czujnik_wilgotnosci_zewnetrzny <= 0 THEN
       "Wejscia_PLC".czujnik_wilgotnosci_zewnetrzny := 0;
   END_IF;
   IF "Wejscia_PLC".Wewnetrzny_czujnik_CO2 <= 0 THEN "Wejscia_PLC".Wewnetrzny_czujnik_CO2 := 0; END_IF;
   IF "Wejscia_PLC".Zewnetrzny_czujnik_CO2 <= 0 THEN "Wejscia_PLC".Zewnetrzny_czujnik_CO2 := 0; END_IF;
   IF "Wejscia_PLC".Czujnik_natezenia_swiatła <= 0 THEN "Wejscia_PLC".Czujnik_natezenia_swiatła := 0; END_IF;
   IF "Wejscia_PLC".Stopien_zasloniecia_rolet >= 100 THEN
       "Wejscia_PLC".Stopien_zasloniecia_rolet := 100;
   END_IF;
   IF "Wejscia_PLC".Stopien_zasloniecia_rolet <= 0 THEN "Wejscia_PLC".Stopien_zasloniecia_rolet := 0; END_IF;
   IF "Wejscia_PLC".Temperatura_zewnetrzna >= 50.0 THEN "Wejscia_PLC".Temperatura_zewnetrzna := 50.0; END_IF;
   IF "Wejscia_PLC".Temperatura_wewnetrzna >= 50.0 THEN "Wejscia_PLC".Temperatura_wewnetrzna := 50.0; END_IF;
   IF "Siłownik_okien_otwieranie" AND ("Wejscia_PLC".Temperatura_zewnetrzna >= "Wejscia_PLC".Temperatura_wewnetrzna) THEN
       "Wejscia_PLC".Temperatura_wewnetrzna := "Wejscia_PLC".Temperatura_zewnetrzna;
   END_IF;
   IF "Wejscia_PLC".Temperatura_wewnetrzna <= 0.0 THEN "Wejscia_PLC".Temperatura_wewnetrzna := 0.0; END_IF;
END_REGION

REGION Network 20: symulacja predkosci wiatru
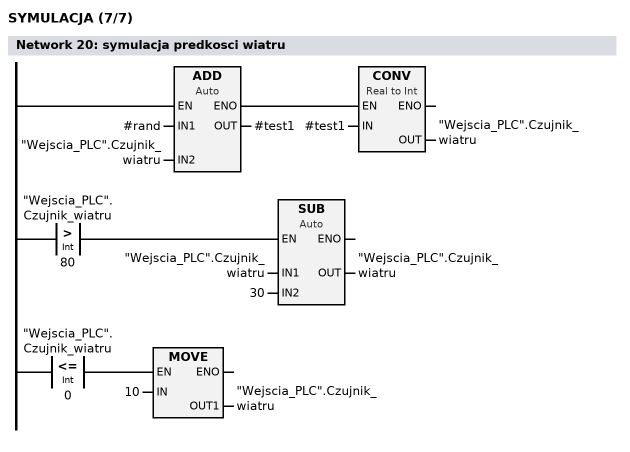
   RUNG wire#powerrail
      { S7_GenerateENO := "TRUE" } Add(in1 := #rand, in2 := "Wejscia_PLC".Czujnik_wiatru, out => #test1)
      { S7_Templates := "[SrcType := Real, DestType := Int]"; S7_GenerateENO := "TRUE" } Convert(in := #test1, out => "Wejscia_PLC".Czujnik_wiatru)
   END_RUNG
   RUNG wire#powerrail
      { S7_Templates := "SrcType := Int" } GT_Contact(in1 := "Wejscia_PLC".Czujnik_wiatru, in2 := 80)
      { S7_GenerateENO := "TRUE" } Sub(in1 := "Wejscia_PLC".Czujnik_wiatru, in2 := 30, out => "Wejscia_PLC".Czujnik_wiatru)
   END_RUNG
   RUNG wire#powerrail
      { S7_Templates := "SrcType := Int" } LE_Contact(in1 := "Wejscia_PLC".Czujnik_wiatru, in2 := 0)
      { S7_GenerateENO := "TRUE" } Move(in := 10, out1 => "Wejscia_PLC".Czujnik_wiatru)
   END_RUNG
   // the same network as SCL:
   // ENO of a box is taken as its EN; it also drops when the box reports an error
   #test1 := #rand + "Wejscia_PLC".Czujnik_wiatru;
   "Wejscia_PLC".Czujnik_wiatru := REAL_TO_INT(#test1);
   IF "Wejscia_PLC".Czujnik_wiatru > 80 THEN
       "Wejscia_PLC".Czujnik_wiatru := "Wejscia_PLC".Czujnik_wiatru - 30;
   END_IF;
   IF "Wejscia_PLC".Czujnik_wiatru <= 0 THEN "Wejscia_PLC".Czujnik_wiatru := 10; END_IF;
END_REGION
END_FUNCTION

ORGANIZATION_BLOCK "Main"   // OB1, LAD, ProgramCycle
TITLE = "Main Program Sweep (Cycle)"
{ S7_Optimized_Access := 'TRUE' }
VERSION : 0.1
   VAR_INPUT
      Initial_Call : Bool;   // Initial call of this OB
      Remanence : Bool;   // =True, if remanent data are available
   END_VAR
   VAR_TEMP
      err : Int;
   END_VAR
   VAR_TEMP   // added for the SCL form of the ladder/FBD networks
      _w1 : Bool;
   END_VAR
BEGIN

REGION Network 1
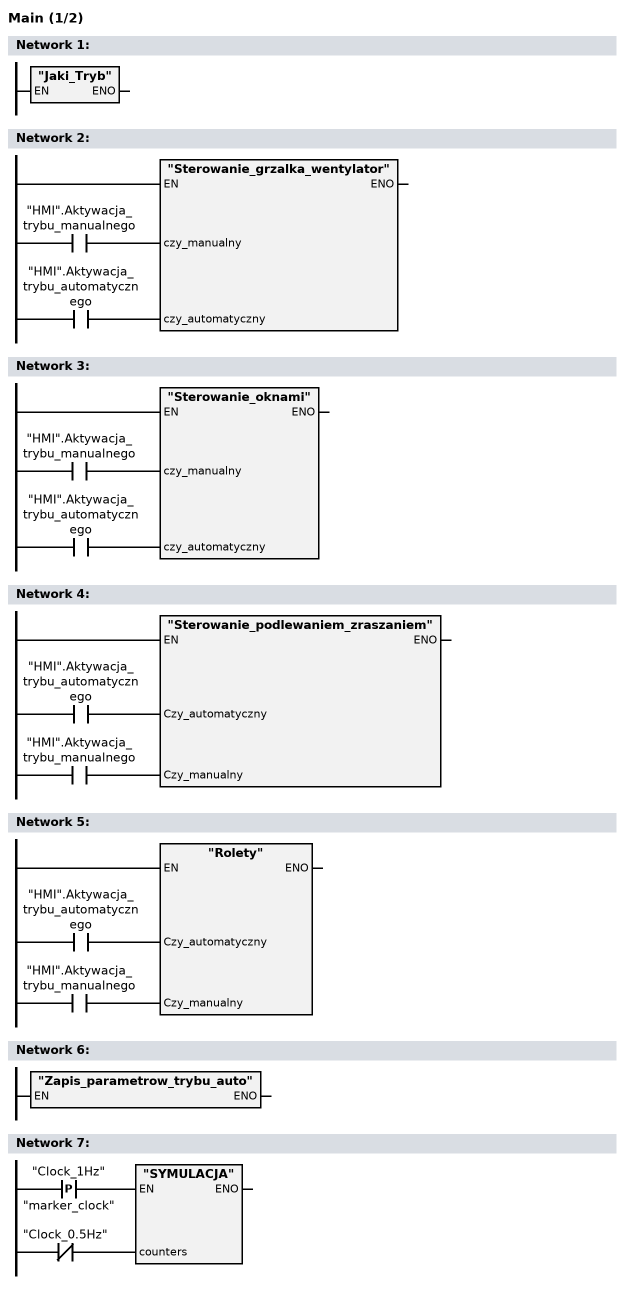
   RUNG wire#powerrail
      "Jaki_Tryb"()
   END_RUNG
   // the same network as SCL:
   "Jaki_Tryb"();
END_REGION

REGION Network 2
   RUNG wire#powerrail
      "Sterowanie_grzalka_wentylator"(czy_manualny := wire#w1, czy_automatyczny := wire#w2)
   END_RUNG
   RUNG wire#powerrail
      Contact( "HMI".Aktywacja_trybu_manualnego )
   END_RUNG wire#w1
   RUNG wire#powerrail
      Contact( "HMI".Aktywacja_trybu_automatycznego )
   END_RUNG wire#w2
   // the same network as SCL:
   "Sterowanie_grzalka_wentylator"(czy_manualny := "HMI".Aktywacja_trybu_manualnego,
                           czy_automatyczny := "HMI".Aktywacja_trybu_automatycznego);
END_REGION

REGION Network 3
   RUNG wire#powerrail
      "Sterowanie_oknami"(czy_manualny := wire#w1, czy_automatyczny := wire#w2)
   END_RUNG
   RUNG wire#powerrail
      Contact( "HMI".Aktywacja_trybu_manualnego )
   END_RUNG wire#w1
   RUNG wire#powerrail
      Contact( "HMI".Aktywacja_trybu_automatycznego )
   END_RUNG wire#w2
   // the same network as SCL:
   "Sterowanie_oknami"(czy_manualny := "HMI".Aktywacja_trybu_manualnego,
                       czy_automatyczny := "HMI".Aktywacja_trybu_automatycznego);
END_REGION

REGION Network 4
   RUNG wire#powerrail
      "Sterowanie_podlewaniem_zraszaniem"(Czy_automatyczny := wire#w1, Czy_manualny := wire#w2)
   END_RUNG
   RUNG wire#powerrail
      Contact( "HMI".Aktywacja_trybu_automatycznego )
   END_RUNG wire#w1
   RUNG wire#powerrail
      Contact( "HMI".Aktywacja_trybu_manualnego )
   END_RUNG wire#w2
   // the same network as SCL:
   "Sterowanie_podlewaniem_zraszaniem"(Czy_automatyczny := "HMI".Aktywacja_trybu_automatycznego,
                           Czy_manualny := "HMI".Aktywacja_trybu_manualnego);
END_REGION

REGION Network 5
   RUNG wire#powerrail
      "Rolety"(Czy_automatyczny := wire#w1, Czy_manualny := wire#w2)
   END_RUNG
   RUNG wire#powerrail
      Contact( "HMI".Aktywacja_trybu_automatycznego )
   END_RUNG wire#w1
   RUNG wire#powerrail
      Contact( "HMI".Aktywacja_trybu_manualnego )
   END_RUNG wire#w2
   // the same network as SCL:
   "Rolety"(Czy_automatyczny := "HMI".Aktywacja_trybu_automatycznego,
            Czy_manualny := "HMI".Aktywacja_trybu_manualnego);
END_REGION

REGION Network 6
   RUNG wire#powerrail
      "Zapis_parametrow_trybu_auto"()
   END_RUNG
   // the same network as SCL:
   "Zapis_parametrow_trybu_auto"();
END_REGION

REGION Network 7
   RUNG wire#powerrail
      P_Contact(operand := "Clock_1Hz", bit := "marker_clock")
      "SYMULACJA"(counters := wire#w1)
   END_RUNG
   RUNG wire#powerrail
      I_Contact( "Clock_0.5Hz" )
   END_RUNG wire#w1
   // the same network as SCL:
   #_w1 := "Clock_1Hz" AND NOT "marker_clock";   // rising edge of "Clock_1Hz"
   "marker_clock" := "Clock_1Hz";
   IF #_w1 THEN "SYMULACJA"(counters := NOT "Clock_0.5Hz"); END_IF;
END_REGION

REGION Network 8
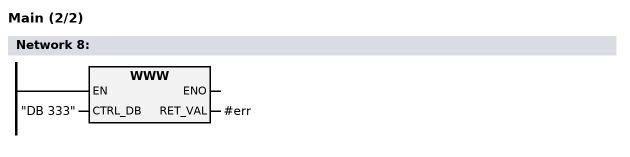
   #err := WWW(CTRL_DB := "DB 333");
END_REGION
END_ORGANIZATION_BLOCK

// folder: Archiwizacja_parametrow

FUNCTION "Archiwizacja_parametrow" : Void   // FC2, LAD
{ S7_Optimized_Access := 'TRUE' }
VERSION : 0.1
// Zapis parametrów do bloku DB odbywa się co pół godziny. Po uruchomieniu sterownika pierwszy zapis nie odbywa się od razu, aby wykres nie przedstawiał parametrów, które nie były jeszcze regulowane. Oczytane watosci zapisywane są w tablicach w bloku DB.
   VAR CONSTANT
      iterator : Int := 0;
   END_VAR
   VAR_TEMP   // added for the SCL form of the ladder/FBD networks
      _w1 : Bool;
   END_VAR
BEGIN

REGION Network 1
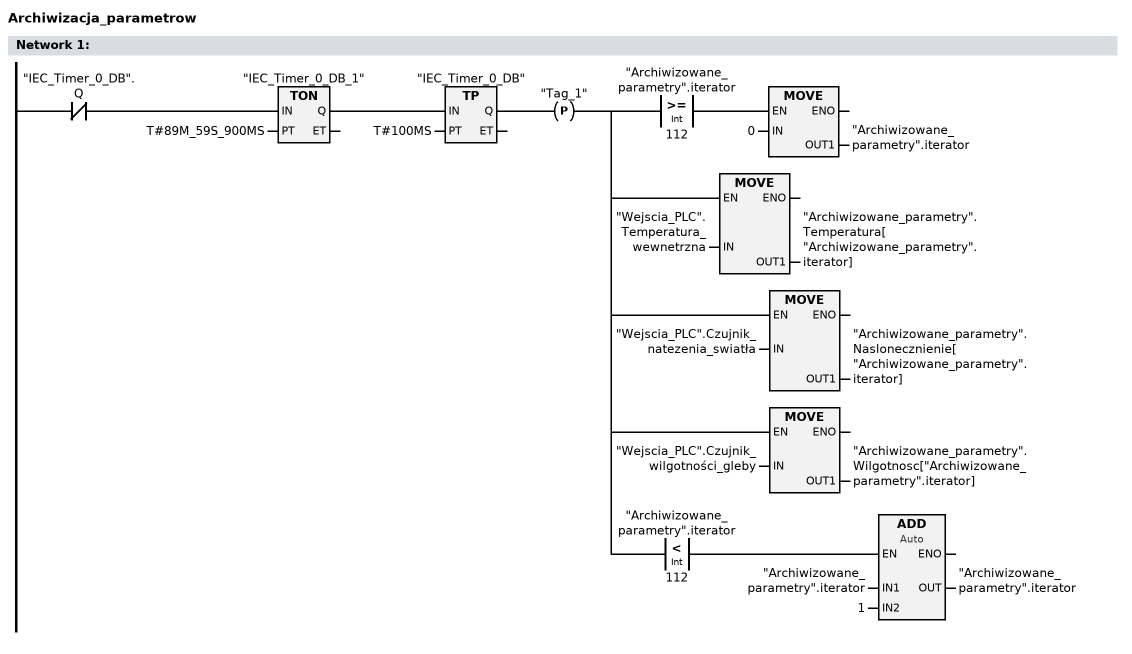
   "IEC_Timer_0_DB_1".TON(IN := NOT "IEC_Timer_0_DB".Q, PT := T#89M_59S_900MS);
   "IEC_Timer_0_DB".TP(IN := "IEC_Timer_0_DB_1".Q, PT := T#100MS);
   #_w1 := "IEC_Timer_0_DB".Q AND NOT "Tag_1";   // rising edge
   "Tag_1" := "IEC_Timer_0_DB".Q;
   IF #_w1 AND ("Archiwizowane_parametry".iterator >= 112) THEN
       "Archiwizowane_parametry".iterator := 0;
   END_IF;
   IF #_w1 THEN
       "Archiwizowane_parametry".Temperatura["Archiwizowane_parametry".iterator] := "Wejscia_PLC".Temperatura_wewnetrzna;
       "Archiwizowane_parametry".Naslonecznienie["Archiwizowane_parametry".iterator] := "Wejscia_PLC".Czujnik_natezenia_swiatła;
       "Archiwizowane_parametry".Wilgotnosc["Archiwizowane_parametry".iterator] := "Wejscia_PLC".Czujnik_wilgotności_gleby;
   END_IF;
   IF #_w1 AND ("Archiwizowane_parametry".iterator < 112) THEN
       "Archiwizowane_parametry".iterator := "Archiwizowane_parametry".iterator + 1;
   END_IF;
END_REGION
END_FUNCTION

// folder: LGF/4 Math operations

FUNCTION "LGF_RandomRange_Real" : Real   // FC10014, SCL
TITLE = LGF_RandomRange_Real
{ S7_Optimized_Access := 'TRUE' }
AUTHOR : Siemens_Digital_Industries
FAMILY : LGF
NAME : LGF_RandomRange_Real
// This function generates random numbers in defined limits (Datatype Real)
   VAR_INPUT
      minValue : Real;   // minimal Value random can reach / Minimum value of the range of the random number
      maxValue : Real;   // maximal Value random can reach / Maximum value of the range of the random number
   END_VAR
   VAR_OUTPUT
      error : Bool;   // Error if true
      status : Word;   // Status of the function
      subfunctionStatus : Word;   // Status or return value of called FB's, FCs and system blocks
   END_VAR
   VAR_TEMP
      tempTime : DTL;   // System time
      tempNanoSecondInDWord : DWord;   // UDINT converted to DWORD for access to individual bytes
      tempTimeStatus : Word;   // Status of the instruction RD_SYS_T
      tempRandomValue : DWord;   // Random-start-value
      tempNormReal : Real;   // normalized value
   END_VAR
   // Ret_Val : Returns random Real number in predefined range
   VAR CONSTANT
      ZERO : Real := 0.0;   // Zero value in case of error
      MAX_UDINT : UDInt := 4294967295;   // Maximum UDINT value
      SUB_STATUS_NO_ERROR : Word := 16#0000;   // Status: sub function call ends without error
      STATUS_FINISHED_NO_ERROR : Word := 16#0000;   // Status: Execution finished without errors
      ERR_MAX_LESS_MIN : Word := 16#8200;   // Error: The maximum limit number is smaller than the minimum limit number
      ERR_RD_SYS_T : Word := 16#8600;   // Error: System function Read system time returned an error
   END_VAR
BEGIN
   REGION Block info header
     //=============================================================================
     // SIEMENS AG / (c)Copyright 2017
     //-----------------------------------------------------------------------------
     // Title:            LGF_RandomRange_Real
     // Comment/Function: This function generates random numbers in defined limits (Datatype Real)
     // Library/Family:   LGF(Library General Functions)
     // Author:           Siemens Digital Industry Support
     // Tested with:      S7-PLCSIM Advanced V2.0 SP1
     // Engineering:      TIA Portal V15 Update 2
     // Restrictions:     ENO disabled - error handling done by error and status
     // Requirements:     PLC (S7-1200 / S7-1500)
     //-------------------------------------------------------------------------------
     // Change log table:
     // Version  | Date       | Expert in charge       | Changes applied
     //----------|------------|------------------------|------------------------------
     // 01.00.00 19.08.2015  Siemens Industry Online Support
     //                      First released version
     // 01.00.01 02.01.2017  Siemens Industry Online Support
     //                      Upgrade: TIA Portal V14 Update 1
     // 01.00.02 02.03.2017  Siemens Industry Online Support
     //                      Bugfix: FC number
     // 01.00.03 17.08.2018  Siemens Industry Online Support
     //                      Upgrade: TIA V15 Update 2
     // 01.00.04 23.11.2018  Siemens Industry Online Support
     //                      Upgrade: TIA V15.1
     // 01.01.00 13.11.2019  Siemens Industry Presales Support
     //                      Renamed from "LGF_RandomReal" to "LGF_RandomRange_Real"
     //                      Regions, commens and costants are added
     // 03.00.00 23.04.2020  Siemens Industry Support
     //                      Set version to V3.0.0, harmonize the version of the whole library
     //=============================================================================
   END_REGION

   REGION Validation
     // Check if the maximal Value is less than the minimal value
     IF (#minValue > #maxValue) THEN
       #error := true;
       #status := #ERR_MAX_LESS_MIN;
       #subfunctionStatus := #SUB_STATUS_NO_ERROR;
       #LGF_RandomRange_Real := #ZERO;
       RETURN;
     END_IF;

     // Read system time
     #tempTimeStatus := INT_TO_WORD(RD_SYS_T(#tempTime));

     // Check return variable for error
     IF (#tempTimeStatus <> #SUB_STATUS_NO_ERROR) THEN
       #error := true;
       #status := #ERR_RD_SYS_T;
       #subfunctionStatus := #tempTimeStatus;
       #LGF_RandomRange_Real := #ZERO;
       RETURN;
     END_IF;
   END_REGION

   REGION Calculating random number
     // Converting to double word so individual bytes can be addressed
     #tempNanoSecondInDWord := UDINT_TO_DWORD(#tempTime.NANOSECOND);

     // Calculate a random-start-value depending on the time
     #tempRandomValue.%B3 := #tempNanoSecondInDWord.%B0;
     #tempRandomValue.%B2 := #tempNanoSecondInDWord.%B1;
     #tempRandomValue.%B1 := #tempNanoSecondInDWord.%B2;
     #tempRandomValue.%B0 := #tempNanoSecondInDWord.%B3;

     // Norm the calculated random number: 0.0 <= #tempNormReal <= 1.0
     #tempNormReal := UDINT_TO_REAL(DWORD_TO_UDINT(#tempRandomValue)) / UDINT_TO_REAL(#MAX_UDINT);

     // Scale the tempNormReal to be in the range of maxValue and minValue
     #LGF_RandomRange_Real := ((#tempNormReal * (#maxValue - #minValue) + (#minValue)));

     #error := false;
     #status := #STATUS_FINISHED_NO_ERROR;
     #subfunctionStatus := #SUB_STATUS_NO_ERROR;
     // ENO mechanism is not used
     ENO := TRUE;
   END_REGION
END_FUNCTION

// ===== PLC "PLC_do_symulacji"  CPU 1214C AC/DC/Rly =====

VAR_GLOBAL   // PLC tag table "Default tag table"
   "Tag_1" AT %M0.0 : Bool;
   "System_Byte" AT %MB1 : Byte;
   "FirstScan" AT %M1.0 : Bool;
   "DiagStatusUpdate" AT %M1.1 : Bool;
   "AlwaysTRUE" AT %M1.2 : Bool;
   "AlwaysFALSE" AT %M1.3 : Bool;
   "Tag_2" AT %M0.1 : Bool;
   "Clock_Byte" AT %MB30 : Byte;
   "Clock_10Hz" AT %M30.0 : Bool;
   "Clock_5Hz" AT %M30.1 : Bool;
   "Clock_2.5Hz" AT %M30.2 : Bool;
   "Clock_2Hz" AT %M30.3 : Bool;
   "Clock_1.25Hz" AT %M30.4 : Bool;
   "Clock_1Hz" AT %M30.5 : Bool;
   "Clock_0.625Hz" AT %M30.6 : Bool;
   "Clock_0.5Hz" AT %M30.7 : Bool;
   "marker_clock" AT %M0.2 : Bool;
   "marker_counter" AT %M0.3 : Bool;
   "wartosc_rolet_sym" AT %MW2 : Int;
   "swiatlo_bez_rolet" AT %MW4 : Int;
   "Alarm_active" AT %M6.0 : Bool;
END_VAR

VAR_GLOBAL   // PLC tag table "wyjscia"
   "Grzałka" AT %Q0.0 : Bool;
   "Wentylator" AT %Q0.1 : Bool;
   "Pompa_zraszacze" AT %Q0.2 : Bool;   // Pompa zraszaczy, które odpowiadają za wilgotność powietrza w szklarni
   "Rolety_zamykanie" AT %Q0.4 : Bool;
   "Alarm_ostrzegwaczy" AT %Q0.5 : Bool;
   "Siłownik_okien_otwieranie" AT %Q0.6 : Bool;
   "Siłownik_okien_zamykanie" AT %Q0.7 : Bool;
   "Rolety_otwieranie" AT %Q0.3 : Bool;
   "Pompa_podlewanie" AT %Q1.0 : Bool;   // Pompa podlewania kropelkowego, która odpowiada za wilgotność gleby
END_VAR

DATA_BLOCK "Wejscia_PLC"   // DB1
{ S7_Optimized_Access := 'TRUE' }
VERSION : 0.1
   VAR
      Czujnik_wilgotności_powietrza : Int;   // Czujnik wilgotności powietrza w szklarni
      Czujnik_wilgotności_gleby : Int;   // Czujnik wilgotności gleby w szklarni
      Temperatura_wewnetrzna : Real;   // Temperatura wewnątrz szklarni
      Czujnik_natezenia_swiatła : Int;   // Czujnik natężenia światła wewnątrz szklarni
      Czujnik_wiatru : Int;   // Czujnik prędkości wiatru poza szklarnią
      Wewnetrzny_czujnik_CO2 : Int;   // Czujnik stężenia dwutlenku węgla w szklarni
      Stopien_zasloniecia_rolet : Int;   // Stopień zasłonięcia rolet w szklarni (przyjęty przedział 0-100%)
      Temperatura_zewnetrzna : Real;   // Temperatura mierzona na zewnątrz, poza szklarnią. Typ Int, ponieważ nie jest wymagana taka dokładność jak w pomiarze temperatury wewnętrznej.
      Zewnetrzny_czujnik_CO2 : Int;   // Czujnik stężenia dwutlenku węgla poza szklarnią
      czujnik_wilgotnosci_zewnetrzny : Int := 50;   // Potrzebny w ramach symulacji realnych warunkow
   END_VAR
BEGIN
END_DATA_BLOCK

DATA_BLOCK "HMI"   // DB2
{ S7_Optimized_Access := 'TRUE' }
VERSION : 0.1
   VAR
      nazwa_receptury : String;
      System_okien_auto : Bool;   // Wł/wył system okien w trybie automatycznym
      Przycisk_zraszacze_manual : Bool;   // Przycisk pompy zraszaczy w trybie manualnym
      Przycisk_podlewanie_manual : Bool;   // Przycisk pompy podlewania w trybie manualnym
      Przycisk_grzanie_manual : Bool;   // Przycisk grzałki w trybie manualnym
      Przycisk_wentylacja_manual : Bool;   // Przycisk wentylacji w trybie manualnym
      Otwarcie_okien_manual : Bool;   // Ustawiony w trybie manualnym otwarcie okien
      Stopien_zasloniecia_rolet_manual : Int;   // Ustawiony w trybie manualnym stopień zasłonięcia rolet
      Temperatura_auto : Real := 22.0;   // Nastawiona temeratura w trybie automatycznym
      Naslonecznienie_auto : Int := 1000;   // Nastawiona wartość nasłonecznienia w trybie automatycznym
      Wilgotnosc_powietrza_auto : Int := 50;   // Nastawiona wartość wilgotności powietrza w trybie automatycznym
      Poziom_CO2_auto : Int := 800;   // Nastawiona wartość stężenia CO2 w trybie automatycznym
      Wilgotnosc_gleby_auto : Int := 60;   // Nastawiona wartość wilgotności gleby w trybie automatycznym
      Przycisk_zatwierdz_auto : Bool;   // Przycisk zatwierdzający wcześniej wybrane ustawienia trybu automatycznego
      Przycisk_zatwierdz_zapis_receptury : Bool;   // Przycisk zatwierdzający wcześniej wybrane ustawienia trybu zapisania receptury
      Przycisk_zatwierdz_wybor_receptury : Bool;   // Przycisk zatwierdzający wcześniej wybrane ustawienia trybu receptury
      Numer_ekranu_HMI : Int;   // Numer aktualnie otwartego ekranu w HMI
      Aktywacja_trybu_manualnego : Bool;
      Aktywacja_trybu_automatycznego : Bool;
      Aktywacja_trybu_Receptur : Bool;
      Aktywacja_trybu_zapis_Receptur : Bool;
      Reset_Trybow : Bool;
   END_VAR
BEGIN
END_DATA_BLOCK

DATA_BLOCK "Tryb_auto_parametry"   // DB7
{ S7_Optimized_Access := 'TRUE' }
VERSION : 0.1
   VAR
      Temperatura : Real;
      Naslonecznienie : Int;
      Wilgotnosc_powietrza : Int;
      Wilgotnosc_gleby : Int;
      System_okien : Bool;
      Stezenie_co2 : Int;
   END_VAR
BEGIN
END_DATA_BLOCK

DATA_BLOCK "Alarmy"   // DB9
{ S7_Optimized_Access := 'TRUE' }
VERSION : 0.1
   VAR
      Warning_niska_temp : String := 'Zbyt niska wartość temperatury utrzymuje się długi czas. Sprawdź grzałkę lub czujnik temperatury.';   // Treść ostrzeżenia wyświetlającego się, gdy temperatura przez długi czas mieści się poniżej wymaganej wartości
      Warning_niska_temp_1 : Bool;
      Warning_wysoka_temp : String := 'Zbyt wysoka wartość temperatury utrzymuje się długi czas. Sprawdź wentylator lub czujnik temperatury.';   // Treść ostrzeżenia wyświetlającego się, gdy temperatura przez długi czas mieści się powyżej wymaganej wartości
      Warning_wysoka_temp_1 : Bool;
      Warning_nieprawidlowe_CO2 : String := 'Stężenie CO2 w zklarni przez długi czas nie osiąga prawidłowych wartości!';   // Treść ostrzeżenia wyświetlającego się, gdy stężenie CO2 w szklarni nie mieści się przez długi czas w wymaganym zakresie
      Warning_nieprawidlowe_CO2_1 : Bool;
      Blad_zbyt_wysokie_CO2 : String := 'Stężenie CO2 w szklarni ma zbyt wysoki poziom. Należy otworzyć okna, uruchomić wentylator lub podjąć inn działania.';   // Treść błędu wyświetlającego się, gdy stężenie CO2 w szklarni ma zbyt wysoki poziom.
      Blad_zbyt_wysokie_CO2_1 : Bool;
   END_VAR
BEGIN
END_DATA_BLOCK

// folder: Archiwizacja_parametrow

DATA_BLOCK "Archiwizowane_parametry"   // DB4
{ S7_Optimized_Access := 'TRUE' }
VERSION : 0.1
   VAR
      Temperatura : Array[0..111] of Real;
      Wilgotnosc : Array[0..111] of Int;
      Naslonecznienie : Array[0..111] of Int;
      iterator : Int := 0;   // Iterator służący do zapisu danych w odpowiednich komórkach tablicy.
   END_VAR
BEGIN
   Naslonecznienie[0] := 0;
   Naslonecznienie[1] := 0;
END_DATA_BLOCK

// folder: System blocks/Program resources

DATA_BLOCK "IEC_Counter_0_DB_1"   // DB3
{ S7_Optimized_Access := 'TRUE' }
AUTHOR : Simatic
FAMILY : IEC
NAME : CNTR
VERSION : 1.0
// stored: InstanceOfName IEC_COUNTER
"IEC_COUNTER"
BEGIN
END_DATA_BLOCK

DATA_BLOCK "IEC_Timer_0_DB"   // DB5
{ S7_Optimized_Access := 'TRUE' }
AUTHOR : Simatic
FAMILY : IEC
NAME : IEC_TMR
VERSION : 1.0
// stored: InstanceOfName IEC_TIMER
"IEC_TIMER"
BEGIN
END_DATA_BLOCK

DATA_BLOCK "IEC_Timer_0_DB_1"   // DB6
{ S7_Optimized_Access := 'TRUE' }
AUTHOR : Simatic
FAMILY : IEC
NAME : IEC_TMR
VERSION : 1.0
// stored: InstanceOfName IEC_TIMER
"IEC_TIMER"
BEGIN
END_DATA_BLOCK

DATA_BLOCK "IEC_Timer_0_DB_2"   // DB8
{ S7_Optimized_Access := 'TRUE' }
AUTHOR : Simatic
FAMILY : IEC
NAME : IEC_TMR
VERSION : 1.0
// stored: InstanceOfName IEC_TIMER
"IEC_TIMER"
BEGIN
END_DATA_BLOCK

DATA_BLOCK "IEC_Timer_0_DB_5"   // DB10
{ S7_Optimized_Access := 'TRUE' }
AUTHOR : Simatic
FAMILY : IEC
NAME : IEC_TMR
VERSION : 1.0
// stored: InstanceOfName IEC_TIMER
"IEC_TIMER"
BEGIN
END_DATA_BLOCK

DATA_BLOCK "IEC_Timer_0_DB_3"   // DB11
{ S7_Optimized_Access := 'TRUE' }
AUTHOR : Simatic
FAMILY : IEC
NAME : IEC_TMR
VERSION : 1.0
// stored: InstanceOfName IEC_TIMER
"IEC_TIMER"
BEGIN
END_DATA_BLOCK

DATA_BLOCK "IEC_Counter_0_DB"   // DB12
{ S7_Optimized_Access := 'TRUE' }
AUTHOR : Simatic
FAMILY : IEC
NAME : CNTR
VERSION : 1.0
// stored: InstanceOfName IEC_COUNTER
"IEC_COUNTER"
BEGIN
END_DATA_BLOCK

DATA_BLOCK "IEC_Counter_0_DB_2"   // DB13
{ S7_Optimized_Access := 'TRUE' }
AUTHOR : Simatic
FAMILY : IEC
NAME : CNTR
VERSION : 1.0
// stored: InstanceOfName IEC_COUNTER
"IEC_COUNTER"
BEGIN
END_DATA_BLOCK

// folder: (top level)

FUNCTION "Rolety" : Void   // FC1, LAD
{ S7_Optimized_Access := 'TRUE' }
VERSION : 0.1
   VAR_INPUT
      Czy_automatyczny : Bool;
      Czy_manualny : Bool;
   END_VAR
BEGIN

REGION Network 1: Warunki otwierania rolet w trybie automatycznym i manualnym
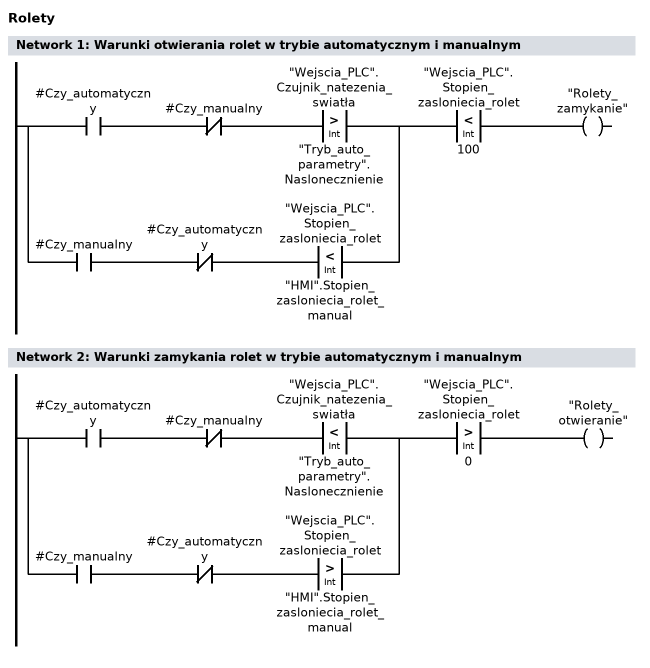
   RUNG wire#powerrail
      Contact( #Czy_automatyczny )
      I_Contact( #Czy_manualny )
      { S7_Templates := "SrcType := Int" } GT_Contact(in1 := "Wejscia_PLC".Czujnik_natezenia_swiatła, in2 := "Tryb_auto_parametry".Naslonecznienie)
      wire#w1
      { S7_Templates := "SrcType := Int" } LT_Contact(in1 := "Wejscia_PLC".Stopien_zasloniecia_rolet, in2 := 100)
      Coil( "Rolety_zamykanie" )
   END_RUNG
   RUNG wire#powerrail
      Contact( #Czy_manualny )
      I_Contact( #Czy_automatyczny )
      { S7_Templates := "SrcType := Int" } LT_Contact(in1 := "Wejscia_PLC".Stopien_zasloniecia_rolet, in2 := "HMI".Stopien_zasloniecia_rolet_manual)
   END_RUNG wire#w1
   // the same network as SCL:
   "Rolety_zamykanie" := ((#Czy_automatyczny AND NOT #Czy_manualny AND ("Wejscia_PLC".Czujnik_natezenia_swiatła > "Tryb_auto_parametry".Naslonecznienie)) OR (#Czy_manualny AND NOT #Czy_automatyczny AND ("Wejscia_PLC".Stopien_zasloniecia_rolet < "HMI".Stopien_zasloniecia_rolet_manual))) AND ("Wejscia_PLC".Stopien_zasloniecia_rolet < 100);
END_REGION

REGION Network 2: Warunki zamykania rolet w trybie automatycznym i manualnym
   RUNG wire#powerrail
      Contact( #Czy_automatyczny )
      I_Contact( #Czy_manualny )
      { S7_Templates := "SrcType := Int" } LT_Contact(in1 := "Wejscia_PLC".Czujnik_natezenia_swiatła, in2 := "Tryb_auto_parametry".Naslonecznienie)
      wire#w1
      { S7_Templates := "SrcType := Int" } GT_Contact(in1 := "Wejscia_PLC".Stopien_zasloniecia_rolet, in2 := 0)
      Coil( "Rolety_otwieranie" )
   END_RUNG
   RUNG wire#powerrail
      Contact( #Czy_manualny )
      I_Contact( #Czy_automatyczny )
      { S7_Templates := "SrcType := Int" } GT_Contact(in1 := "Wejscia_PLC".Stopien_zasloniecia_rolet, in2 := "HMI".Stopien_zasloniecia_rolet_manual)
   END_RUNG wire#w1
   // the same network as SCL:
   "Rolety_otwieranie" := ((#Czy_automatyczny AND NOT #Czy_manualny AND ("Wejscia_PLC".Czujnik_natezenia_swiatła < "Tryb_auto_parametry".Naslonecznienie)) OR (#Czy_manualny AND NOT #Czy_automatyczny AND ("Wejscia_PLC".Stopien_zasloniecia_rolet > "HMI".Stopien_zasloniecia_rolet_manual))) AND ("Wejscia_PLC".Stopien_zasloniecia_rolet > 0);
END_REGION
END_FUNCTION

FUNCTION "Sterowanie_grzalka_wentylator" : Void   // FC3, LAD
{ S7_Optimized_Access := 'TRUE' }
VERSION : 0.1
   VAR_INPUT
      czy_manualny : Bool;
      czy_automatyczny : Bool;
   END_VAR
   VAR_TEMP
      Histereza_minus : Real;   // Wartość zadanej temperatury zmieniona o dolną wartość hiterezy
      Histereza_plus : Real;   // Wartość zadanej temperatury zmieniona o górną wartość hiterezy
   END_VAR
   VAR CONSTANT
      Wartosc_histerezy : Real := 1.0;
   END_VAR
   VAR_TEMP   // added for the SCL form of the ladder/FBD networks
      _w1 : Bool;
   END_VAR
BEGIN

REGION Network 1: Sterowanie wentylatorem w trybie automatycznym i manualnym
   // Gdy uruchomiony jest tryb automatyczny, wartość temperatury w szklarni powinna się mieścić w zakresie temperatury nastawionej +- wartość histerezy. Gdy jest ona za wysoka uruchamiany jest wentylator. W trybie manualnym włączany jest on od razu po naciśnięciu przycisku do niego przypisanego.
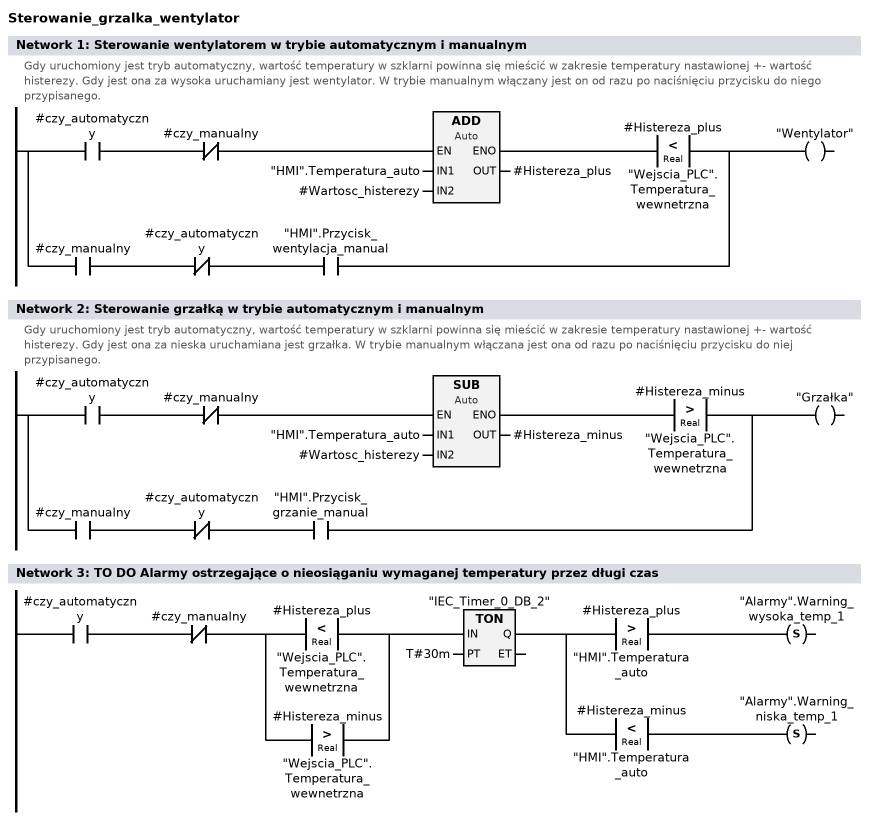
   RUNG wire#powerrail
      Contact( #czy_automatyczny )
      I_Contact( #czy_manualny )
      Add(in1 := "HMI".Temperatura_auto, in2 := #Wartosc_histerezy, out => #Histereza_plus)
      { S7_Templates := "SrcType := Real" } LT_Contact(in1 := #Histereza_plus, in2 := "Wejscia_PLC".Temperatura_wewnetrzna)
      wire#w1
      Coil( "Wentylator" )
   END_RUNG
   RUNG wire#powerrail
      Contact( #czy_manualny )
      I_Contact( #czy_automatyczny )
      Contact( "HMI".Przycisk_wentylacja_manual )
   END_RUNG wire#w1
   // the same network as SCL:
   #_w1 := #czy_automatyczny AND NOT #czy_manualny;
   IF #_w1 THEN #Histereza_plus := "HMI".Temperatura_auto + #Wartosc_histerezy; END_IF;
   "Wentylator" := (#_w1 AND (#Histereza_plus < "Wejscia_PLC".Temperatura_wewnetrzna)) OR (#czy_manualny AND NOT #czy_automatyczny AND "HMI".Przycisk_wentylacja_manual);
END_REGION

REGION Network 2: Sterowanie grzałką w trybie automatycznym i manualnym
   // Gdy uruchomiony jest tryb automatyczny, wartość temperatury w szklarni powinna się mieścić w zakresie temperatury nastawionej +- wartość histerezy. Gdy jest ona za nieska uruchamiana jest grzałka. W trybie manualnym włączana jest ona od razu po naciśnięciu przycisku do niej przypisanego.
   RUNG wire#powerrail
      Contact( #czy_automatyczny )
      I_Contact( #czy_manualny )
      Sub(in1 := "HMI".Temperatura_auto, in2 := #Wartosc_histerezy, out => #Histereza_minus)
      { S7_Templates := "SrcType := Real" } GT_Contact(in1 := #Histereza_minus, in2 := "Wejscia_PLC".Temperatura_wewnetrzna)
      wire#w1
      Coil( "Grzałka" )
   END_RUNG
   RUNG wire#powerrail
      Contact( #czy_manualny )
      I_Contact( #czy_automatyczny )
      Contact( "HMI".Przycisk_grzanie_manual )
   END_RUNG wire#w1
   // the same network as SCL:
   #_w1 := #czy_automatyczny AND NOT #czy_manualny;
   IF #_w1 THEN #Histereza_minus := "HMI".Temperatura_auto - #Wartosc_histerezy; END_IF;
   "Grzałka" := (#_w1 AND (#Histereza_minus > "Wejscia_PLC".Temperatura_wewnetrzna)) OR (#czy_manualny AND NOT #czy_automatyczny AND "HMI".Przycisk_grzanie_manual);
END_REGION

REGION Network 3: TO DO Alarmy ostrzegające o nieosiąganiu wymaganej temperatury przez długi czas
   "IEC_Timer_0_DB_2".TON(IN := #czy_automatyczny AND NOT #czy_manualny AND ((#Histereza_plus < "Wejscia_PLC".Temperatura_wewnetrzna) OR (#Histereza_minus > "Wejscia_PLC".Temperatura_wewnetrzna)),
                          PT := T#30m);
   IF "IEC_Timer_0_DB_2".Q AND (#Histereza_plus > "HMI".Temperatura_auto) THEN
       "Alarmy".Warning_wysoka_temp_1 := TRUE;
   END_IF;
   IF "IEC_Timer_0_DB_2".Q AND (#Histereza_minus < "HMI".Temperatura_auto) THEN
       "Alarmy".Warning_niska_temp_1 := TRUE;
   END_IF;
END_REGION
END_FUNCTION

FUNCTION "Zapis_parametrow_trybu_auto" : Void   // FC4, LAD
{ S7_Optimized_Access := 'TRUE' }
VERSION : 0.1
BEGIN

REGION Network 1: Zapis wybranych na HMI parametrów, aby zostały one stałe do kolejnego zatwierdzenia ich zmiany.
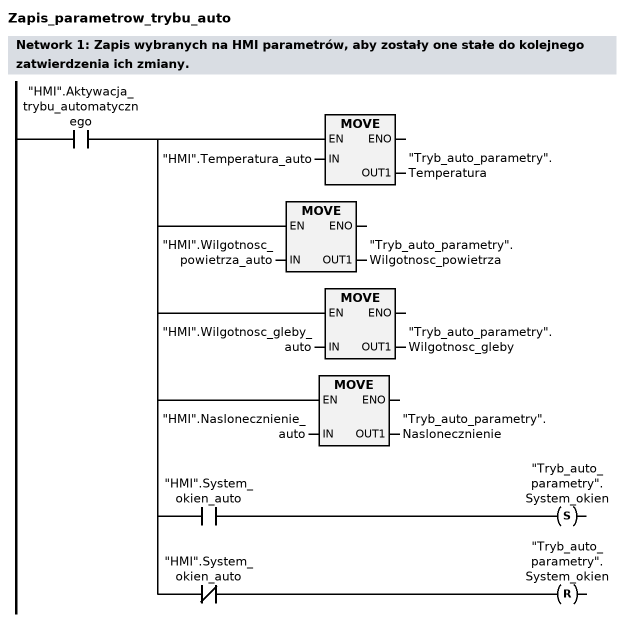
   RUNG wire#powerrail
      Contact( "HMI".Aktywacja_trybu_automatycznego )
      wire#w1
      Move(in := "HMI".Temperatura_auto, out1 => "Tryb_auto_parametry".Temperatura)
   END_RUNG
   RUNG wire#w1
      Move(in := "HMI".Wilgotnosc_powietrza_auto, out1 => "Tryb_auto_parametry".Wilgotnosc_powietrza)
   END_RUNG
   RUNG wire#w1
      Move(in := "HMI".Wilgotnosc_gleby_auto, out1 => "Tryb_auto_parametry".Wilgotnosc_gleby)
   END_RUNG
   RUNG wire#w1
      Move(in := "HMI".Naslonecznienie_auto, out1 => "Tryb_auto_parametry".Naslonecznienie)
   END_RUNG
   RUNG wire#w1
      Contact( "HMI".System_okien_auto )
      S_Coil( "Tryb_auto_parametry".System_okien )
   END_RUNG
   RUNG wire#w1
      I_Contact( "HMI".System_okien_auto )
      R_Coil( "Tryb_auto_parametry".System_okien )
   END_RUNG
   // the same network as SCL:
   IF "HMI".Aktywacja_trybu_automatycznego THEN
       "Tryb_auto_parametry".Temperatura := "HMI".Temperatura_auto;
       "Tryb_auto_parametry".Wilgotnosc_powietrza := "HMI".Wilgotnosc_powietrza_auto;
       "Tryb_auto_parametry".Wilgotnosc_gleby := "HMI".Wilgotnosc_gleby_auto;
       "Tryb_auto_parametry".Naslonecznienie := "HMI".Naslonecznienie_auto;
   END_IF;
   IF "HMI".Aktywacja_trybu_automatycznego AND "HMI".System_okien_auto THEN
       "Tryb_auto_parametry".System_okien := TRUE;
   END_IF;
   IF "HMI".Aktywacja_trybu_automatycznego AND NOT "HMI".System_okien_auto THEN
       "Tryb_auto_parametry".System_okien := FALSE;
   END_IF;
END_REGION
END_FUNCTION

FUNCTION "Jaki_Tryb" : Void   // FC5, LAD
{ S7_Optimized_Access := 'TRUE' }
VERSION : 0.1
BEGIN

REGION Network 1: Reset trybu auto jesli wykryje jakikolwiek inny tryb
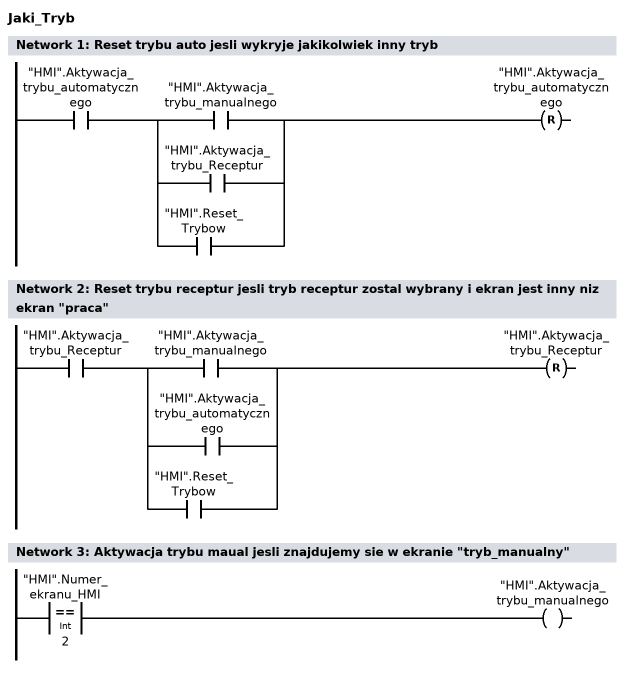
   RUNG wire#powerrail
      Contact( "HMI".Aktywacja_trybu_automatycznego )
      wire#w1
      Contact( "HMI".Aktywacja_trybu_manualnego )
      wire#w2
      R_Coil( "HMI".Aktywacja_trybu_automatycznego )
   END_RUNG
   RUNG wire#w1
      Contact( "HMI".Aktywacja_trybu_Receptur )
   END_RUNG wire#w2
   RUNG wire#w1
      Contact( "HMI".Reset_Trybow )
   END_RUNG wire#w2
   // the same network as SCL:
   IF "HMI".Aktywacja_trybu_automatycznego AND ("HMI".Aktywacja_trybu_manualnego OR "HMI".Aktywacja_trybu_Receptur OR "HMI".Reset_Trybow) THEN
       "HMI".Aktywacja_trybu_automatycznego := FALSE;
   END_IF;
END_REGION

REGION Network 2: Reset trybu receptur jesli tryb receptur zostal wybrany i ekran jest inny niz ekran "praca"
   RUNG wire#powerrail
      Contact( "HMI".Aktywacja_trybu_Receptur )
      wire#w1
      Contact( "HMI".Aktywacja_trybu_manualnego )
      wire#w2
      R_Coil( "HMI".Aktywacja_trybu_Receptur )
   END_RUNG
   RUNG wire#w1
      Contact( "HMI".Aktywacja_trybu_automatycznego )
   END_RUNG wire#w2
   RUNG wire#w1
      Contact( "HMI".Reset_Trybow )
   END_RUNG wire#w2
   // the same network as SCL:
   IF "HMI".Aktywacja_trybu_Receptur AND ("HMI".Aktywacja_trybu_manualnego OR "HMI".Aktywacja_trybu_automatycznego OR "HMI".Reset_Trybow) THEN
       "HMI".Aktywacja_trybu_Receptur := FALSE;
   END_IF;
END_REGION

REGION Network 3: Aktywacja trybu maual jesli znajdujemy sie w ekranie "tryb_manualny"
   RUNG wire#powerrail
      { S7_Templates := "SrcType := Int" } EQ_Contact(in1 := "HMI".Numer_ekranu_HMI, in2 := 2)
      Coil( "HMI".Aktywacja_trybu_manualnego )
   END_RUNG
   // the same network as SCL:
   "HMI".Aktywacja_trybu_manualnego := "HMI".Numer_ekranu_HMI = 2;
END_REGION
END_FUNCTION

FUNCTION "Ograniczanie_wartosci_parametrow" : Void   // FC6, LAD
TITLE = Każdy z poniższych network-ów odpowiada za to, aby po ustawieniu na HMI wartości przekraczajacej dopuszczalną, ta pozostała w wymaganym zakresie.
{ S7_Optimized_Access := 'TRUE' }
VERSION : 0.1
BEGIN

REGION Network 1: Ograniczenie dla wartosci ustawionej temperatury w trybie automatycznym
